KUKA KRL program: MyProgram_333().src

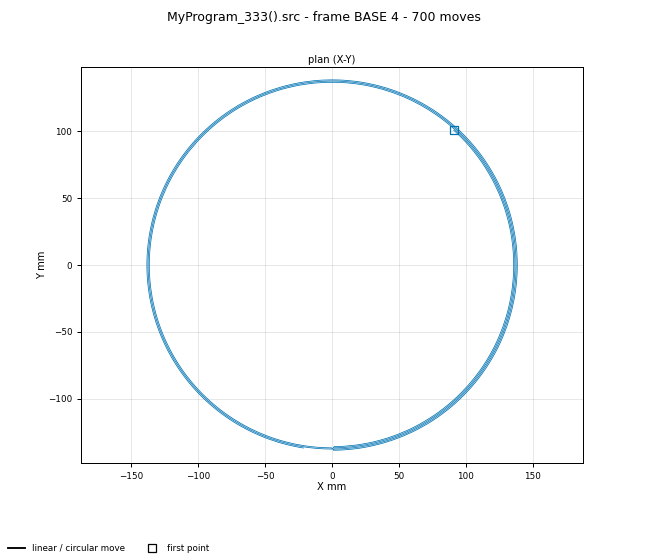
[picture p0: tool path of MyProgram_333().src in frame BASE 4, 700 of 700 moves have a stored position in this frame; points joined in program order, loops and branches not executed]
&ACCESS RVP
&REL 1
&PARAM TEMPLATE = C:\KRC\Roboter\Template\vorgabe
&PARAM EDITMASK = *
DEF MyProgram_333()
; ---- Setting reference (Base) ----
$BASE = BASE_DATA[4]

; --------------------------
; ---- Setting tool (TCP) ----
$TOOL = TOOL_DATA[3]
; --------------------------

$VEL.CP = VEL_APROX_PRINT
Startdeposition()
$VEL.CP = VEL_PRINT
LIN {X 90.8703,Y 100.8423,Z 189,A 47.7987,B 1.7183,C 0.0098,E1 1.8301,E2 406.2079} C_DIS
LIN {X 94.1895,Y 97.749,Z 189,A 46.0059,B 1.7183,C 0.013,E1 1.8337,E2 407.9863} C_DIS
LIN {X 97.3671,Y 94.5838,Z 189,A 44.2321,B 1.7183,C 0.0163,E1 1.8371,E2 409.7463} C_DIS
LIN {X 100.4728,Y 91.2777,Z 189,A 42.4362,B 1.7183,C 0.0197,E1 1.8405,E2 411.5282} C_DIS
LIN {X 103.5335,Y 87.791,Z 189,A 40.6188,B 1.7182,C 0.0232,E1 1.8438,E2 413.3292} C_DIS
LIN {X 106.2609,Y 84.4691,Z 189,A 38.9353,B 1.7182,C 0.0265,E1 1.8467,E2 414.9974} C_DIS
LIN {X 108.9996,Y 80.9045,Z 189,A 37.1372,B 1.7181,C 0.0303,E1 1.8498,E2 416.7841} C_DIS
LIN {X 111.6341,Y 77.2293,Z 189,A 34.7595,B 1.7179,C 0.0378,E1 1.8537,E2 419.2181} C_DIS
LIN {X 114.6999,Y 72.5973,Z 189,A 33.3263,B 1.7179,C 0.0378,E1 1.8557,E2 420.5428} C_DIS
LIN {X 117.6265,Y 67.7532,Z 189,A 31.0653,B 1.7179,C 0.0428,E1 1.8589,E2 422.7891} C_DIS
LIN {X 119.3923,Y 64.5914,Z 189,A 29.4618,B 1.7177,C 0.0471,E1 1.861,E2 424.4021} C_DIS
LIN {X 121.4958,Y 60.5386,Z 189,A 27.7475,B 1.7176,C 0.0506,E1 1.8632,E2 426.091} C_DIS
LIN {X 124.3864,Y 54.3522,Z 189,A 25.1966,B 1.7174,C 0.0559,E1 1.8661,E2 428.6026} C_DIS
LIN {X 125.7898,Y 51.0185,Z 189,A 23.03,B 1.7171,C 0.0642,E1 1.8685,E2 430.8476} C_DIS
LIN {X 127.7963,Y 45.7611,Z 189,A 21.5201,B 1.7171,C 0.0648,E1 1.8698,E2 432.253} C_DIS
LIN {X 128.8823,Y 42.6068,Z 189,A 20.1683,B 1.717,C 0.0681,E1 1.871,E2 433.5984} C_DIS
LIN {X 130.1919,Y 38.4196,Z 189,A 18.4533,B 1.7168,C 0.0722,E1 1.8724,E2 435.2973} C_DIS
LIN {X 131.1658,Y 34.9492,Z 189,A 17.0946,B 1.7167,C 0.0753,E1 1.8734,E2 436.6367} C_DIS
LIN {X 131.9479,Y 31.8698,Z 189,A 15.8155,B 1.7165,C 0.0785,E1 1.8743,E2 437.9086} C_DIS
LIN {X 132.7323,Y 28.4276,Z 189,A 14.4424,B 1.7164,C 0.0818,E1 1.8751,E2 439.268} C_DIS
LIN {X 133.5246,Y 24.4421,Z 189,A 12.701,B 1.7161,C 0.0867,E1 1.876,E2 441.0135} C_DIS
LIN {X 134.3255,Y 19.5645,Z 189,A 10.8763,B 1.7159,C 0.0907,E1 1.8768,E2 442.8067} C_DIS
LIN {X 135.0433,Y 13.7704,Z 189,A 8.4484,B 1.7156,C 0.0974,E1 1.8775,E2 445.2313} C_DIS
LIN {X 135.4898,Y 8.2777,Z 189,A 6.4872,B 1.7153,C 0.1014,E1 1.8779,E2 447.1481} C_DIS
LIN {X 135.6826,Y 4.0405,Z 189,A 4.2707,B 1.7149,C 0.1093,E1 1.8781,E2 449.4189} C_DIS
LIN {X 135.7388,Y -1.1337,Z 189,A 2.8572,B 1.7149,C 0.1101,E1 1.8781,E2 450.7369} C_DIS
LIN {X 135.5285,Y -7.6497,Z 189,A 0.3514,B 1.7144,C 0.1162,E1 1.8779,E2 453.2133} C_DIS
LIN {X 135.2924,Y -11.0499,Z 189,A -1.8109,B 1.7138,C 0.1252,E1 1.8774,E2 455.4679} C_DIS
LIN {X 134.6403,Y -17.266,Z 189,A -3.3061,B 1.7138,C 0.1246,E1 1.8769,E2 456.8201} C_DIS
LIN {X 134.2033,Y -20.386,Z 189,A -4.7668,B 1.7135,C 0.1292,E1 1.8763,E2 458.2983} C_DIS
LIN {X 133.5519,Y -24.2894,Z 189,A -6.2722,B 1.7132,C 0.1327,E1 1.8756,E2 459.7837} C_DIS
LIN {X 132.73,Y -28.4383,Z 189,A -7.9415,B 1.7129,C 0.1368,E1 1.8747,E2 461.4394} C_DIS
LIN {X 131.9479,Y -31.8698,Z 189,A -9.2499,B 1.7126,C 0.1397,E1 1.8739,E2 462.726} C_DIS
LIN {X 131.0873,Y -35.2437,Z 189,A -10.6477,B 1.7124,C 0.1432,E1 1.8729,E2 464.1155} C_DIS
LIN {X 130.1198,Y -38.6657,Z 189,A -12.0307,B 1.7121,C 0.1465,E1 1.8718,E2 465.4844} C_DIS
LIN {X 127.4351,Y -46.763,Z 189,A -15.4685,B 1.7113,C 0.155,E1 1.8688,E2 468.9037} C_DIS
LIN {X 124.5568,Y -53.9582,Z 189,A -18.4307,B 1.7107,C 0.1615,E1 1.8657,E2 471.8281} C_DIS
LIN {X 123.0854,Y -57.2358,Z 189,A -19.8254,B 1.7104,C 0.1646,E1 1.864,E2 473.2081} C_DIS
LIN {X 121.5338,Y -60.4615,Z 189,A -21.1963,B 1.7102,C 0.1675,E1 1.8624,E2 474.5619} C_DIS
LIN {X 119.9443,Y -63.5568,Z 189,A -22.6938,B 1.7098,C 0.1714,E1 1.8604,E2 476.0643} C_DIS
LIN {X 117.629,Y -67.7489,Z 189,A -24.6616,B 1.7093,C 0.1761,E1 1.8577,E2 478.0267} C_DIS
LIN {X 115.5415,Y -71.2508,Z 189,A -26.1596,B 1.709,C 0.1789,E1 1.8556,E2 479.4967} C_DIS
LIN {X 113.1519,Y -74.9881,Z 189,A -28.3044,B 1.7083,C 0.1852,E1 1.8523,E2 481.6786} C_DIS
LIN {X 110.5875,Y -78.7204,Z 189,A -29.805,B 1.7081,C 0.1871,E1 1.8499,E2 483.1268} C_DIS
LIN {X 106.2233,Y -84.5164,Z 189,A -32.1804,B 1.7078,C 0.1897,E1 1.8461,E2 485.4136} C_DIS
LIN {X 101.8169,Y -89.7762,Z 189,A -35.2885,B 1.7069,C 0.1975,E1 1.8404,E2 488.5522} C_DIS
LIN {X 97.0122,Y -94.9477,Z 189,A -37.7383,B 1.7066,C 0.2006,E1 1.8359,E2 490.9338} C_DIS
LIN {X 93.5191,Y -98.3907,Z 189,A -40.0626,B 1.7059,C 0.2065,E1 1.8311,E2 493.2937} C_DIS
LIN {X 89.8066,Y -101.79,Z 189,A -42.5349,B 1.7051,C 0.2129,E1 1.8258,E2 495.8137} C_DIS
LIN {X 85.9282,Y -105.0845,Z 189,A -44.0029,B 1.7051,C 0.2129,E1 1.8229,E2 497.1929} C_DIS
LIN {X 82.7199,Y -107.6287,Z 189,A -46.0103,B 1.7045,C 0.2178,E1 1.8183,E2 499.2389} C_DIS
LIN {X 79.5486,Y -109.9929,Z 189,A -47.3444,B 1.7043,C 0.2189,E1 1.8154,E2 500.5294} C_DIS
LIN {X 76.7274,Y -111.9792,Z 189,A -48.6664,B 1.7041,C 0.2206,E1 1.8124,E2 501.8344} C_DIS
LIN {X 73.1409,Y -114.354,Z 189,A -50.3736,B 1.7038,C 0.2231,E1 1.8084,E2 503.5285} C_DIS
LIN {X 66.1262,Y -118.5492,Z 189,A -53.5982,B 1.7032,C 0.2273,E1 1.8007,E2 506.7253} C_DIS
LIN {X 62.9243,Y -120.2765,Z 189,A -55.0845,B 1.703,C 0.2294,E1 1.7971,E2 508.206} C_DIS
LIN {X 59.426,Y -122.0447,Z 189,A -56.6641,B 1.7027,C 0.2313,E1 1.7931,E2 509.7766} C_DIS
LIN {X 56.28,Y -123.5274,Z 189,A -59.0747,B 1.7017,C 0.2386,E1 1.7867,E2 512.3149} C_DIS
LIN {X 49.5643,Y -126.3702,Z 189,A -60.8954,B 1.7021,C 0.2357,E1 1.7824,E2 513.9687} C_DIS
LIN {X 47.2117,Y -127.2679,Z 189,A -62.1901,B 1.7017,C 0.2382,E1 1.7789,E2 515.2956} C_DIS
LIN {X 42.7243,Y -128.8432,Z 189,A -64.0034,B 1.7016,C 0.2395,E1 1.7741,E2 517.0838} C_DIS
LIN {X 39.4837,Y -129.873,Z 189,A -65.3751,B 1.7014,C 0.2407,E1 1.7705,E2 518.4479} C_DIS
LIN {X 36.0559,Y -130.867,Z 189,A -66.9587,B 1.7011,C 0.2426,E1 1.7662,E2 520.0429} C_DIS
LIN {X 32.0339,Y -131.9083,Z 189,A -68.7073,B 1.7009,C 0.2442,E1 1.7614,E2 521.792} C_DIS
LIN {X 28.2791,Y -132.7644,Z 189,A -70.1338,B 1.7009,C 0.2446,E1 1.7576,E2 523.1924} C_DIS
LIN {X 24.9851,Y -133.424,Z 189,A -71.6086,B 1.7006,C 0.246,E1 1.7535,E2 524.6758} C_DIS
LIN {X 18.2831,Y -134.5059,Z 189,A -74.459,B 1.7004,C 0.2478,E1 1.7456,E2 527.5258} C_DIS
LIN {X 9.6151,Y -135.4017,Z 189,A -77.5536,B 1.7004,C 0.2472,E1 1.7372,E2 530.5429} C_DIS
LIN {X 5.6929,Y -135.6236,Z 189,A -80.0456,B 1.6998,C 0.2516,E1 1.7299,E2 533.1494} C_DIS
LIN {X 1.4833,Y -135.7364,Z 189,A -82.2677,B 1.6995,C 0.254,E1 1.7235,E2 535.4324} C_DIS
LIN {X 1.4833,Y -135.7364,Z 189,A -82.2677,B 1.6995,C 0.254,E1 1.7235,E2 535.4325} C_DIS
Enddeposition()
LIN {X 0.9598,Y -136.6371,Z 189,A -81.4185,B 1.6921,C 0.25,E1 1.7183,E2 534.469} C_DIS
Startdeposition()
$VEL.CP = VEL_PRINT
LIN {X 6.638,Y -136.4804,Z 189,A -78.5202,B 1.6925,C 0.2468,E1 1.7266,E2 531.4984} C_DIS
LIN {X 9.6494,Y -136.3007,Z 189,A -76.4403,B 1.6932,C 0.2424,E1 1.7327,E2 529.3043} C_DIS
LIN {X 16.0925,Y -135.6906,Z 189,A -74.9101,B 1.6926,C 0.2465,E1 1.7365,E2 527.9373} C_DIS
LIN {X 23.1959,Y -134.6601,Z 189,A -71.5532,B 1.6931,C 0.2428,E1 1.746,E2 524.531} C_DIS
LIN {X 26.9,Y -133.9678,Z 189,A -70.1444,B 1.6931,C 0.2424,E1 1.7498,E2 523.1449} C_DIS
LIN {X 30.7402,Y -133.139,Z 189,A -68.4565,B 1.6934,C 0.2408,E1 1.7544,E2 521.4504} C_DIS
LIN {X 34.9207,Y -132.104,Z 189,A -66.772,B 1.6935,C 0.2397,E1 1.7589,E2 519.7815} C_DIS
LIN {X 38.144,Y -131.2095,Z 189,A -65.4425,B 1.6937,C 0.2386,E1 1.7625,E2 518.4613} C_DIS
LIN {X 42.1979,Y -129.9638,Z 189,A -63.4142,B 1.6941,C 0.2354,E1 1.768,E2 516.3972} C_DIS
LIN {X 45.2532,Y -128.9311,Z 189,A -62.2617,B 1.6942,C 0.2349,E1 1.771,E2 515.2714} C_DIS
LIN {X 49.0394,Y -127.539,Z 189,A -60.4045,B 1.6946,C 0.2319,E1 1.7759,E2 513.3902} C_DIS
LIN {X 52.3982,Y -126.1955,Z 189,A -58.8181,B 1.6949,C 0.2296,E1 1.78,E2 511.7931} C_DIS
LIN {X 56.5287,Y -124.4023,Z 189,A -57.4744,B 1.6949,C 0.2301,E1 1.7833,E2 510.5234} C_DIS
LIN {X 60.044,Y -122.7424,Z 189,A -55.8889,B 1.6952,C 0.228,E1 1.7873,E2 508.9428} C_DIS
LIN {X 63.4072,Y -121.0385,Z 189,A -54.4087,B 1.6954,C 0.2262,E1 1.7909,E2 507.4753} C_DIS
LIN {X 67.1839,Y -118.9861,Z 189,A -52.2096,B 1.6961,C 0.2211,E1 1.7965,E2 505.2204} C_DIS
LIN {X 70.9392,Y -116.7862,Z 189,A -50.6757,B 1.6962,C 0.2198,E1 1.8,E2 503.7252} C_DIS
LIN {X 75.7995,Y -113.6916,Z 189,A -48.3467,B 1.6967,C 0.2162,E1 1.8055,E2 501.4064} C_DIS
LIN {X 78.5361,Y -111.8185,Z 189,A -47.1452,B 1.6969,C 0.2149,E1 1.8082,E2 500.2298} C_DIS
LIN {X 82.5681,Y -108.8758,Z 189,A -45.2283,B 1.6972,C 0.2121,E1 1.8124,E2 498.3355} C_DIS
LIN {X 86.127,Y -106.0833,Z 189,A -43.5538,B 1.6975,C 0.2099,E1 1.816,E2 496.6898} C_DIS
LIN {X 89.7935,Y -102.9973,Z 189,A -41.3951,B 1.6981,C 0.205,E1 1.8207,E2 494.5093} C_DIS
LIN {X 93.6526,Y -99.5014,Z 189,A -39.4677,B 1.6984,C 0.2022,E1 1.8246,E2 492.6152} C_DIS
LIN {X 96.9373,Y -96.3041,Z 189,A -37.7525,B 1.6987,C 0.1995,E1 1.8279,E2 490.9265} C_DIS
LIN {X 100.3179,Y -92.7775,Z 189,A -35.4013,B 1.6995,C 0.1931,E1 1.8325,E2 488.5326} C_DIS
LIN {X 103.1234,Y -89.649,Z 189,A -34.1162,B 1.6995,C 0.1923,E1 1.8348,E2 487.3109} C_DIS
LIN {X 105.9837,Y -86.2489,Z 189,A -32.351,B 1.7,C 0.1887,E1 1.8379,E2 485.5575} C_DIS
LIN {X 110.3626,Y -80.5696,Z 189,A -29.6513,B 1.7005,C 0.1838,E1 1.8424,E2 482.897} C_DIS
LIN {X 112.6528,Y -77.3346,Z 189,A -27.7228,B 1.7011,C 0.1781,E1 1.8455,E2 480.9314} C_DIS
LIN {X 114.7002,Y -74.2646,Z 189,A -26.5325,B 1.7013,C 0.1767,E1 1.8473,E2 479.788} C_DIS
LIN {X 117.8288,Y -69.1933,Z 189,A -24.2296,B 1.7018,C 0.1719,E1 1.8506,E2 477.5094} C_DIS
LIN {X 119.9886,Y -65.3764,Z 189,A -22.3737,B 1.7022,C 0.1671,E1 1.8531,E2 475.6498} C_DIS
LIN {X 122.2789,Y -60.9836,Z 189,A -20.5833,B 1.7026,C 0.1638,E1 1.8553,E2 473.8962} C_DIS
LIN {X 123.9248,Y -57.5629,Z 189,A -19.1561,B 1.7028,C 0.1608,E1 1.857,E2 472.4897} C_DIS
LIN {X 125.2805,Y -54.5501,Z 189,A -17.3824,B 1.7034,C 0.1545,E1 1.859,E2 470.6632} C_DIS
LIN {X 127.0806,Y -50.2186,Z 189,A -15.9513,B 1.7036,C 0.1531,E1 1.8604,E2 469.3021} C_DIS
LIN {X 128.2149,Y -47.2469,Z 189,A -13.9405,B 1.7043,C 0.1448,E1 1.8625,E2 467.2002} C_DIS
LIN {X 130.4205,Y -40.7672,Z 189,A -12.0416,B 1.7043,C 0.1439,E1 1.8639,E2 465.4285} C_DIS
LIN {X 131.5275,Y -37.0325,Z 189,A -10.6101,B 1.7046,C 0.1408,E1 1.865,E2 464.0224} C_DIS
LIN {X 132.4351,Y -33.6421,Z 189,A -9.3001,B 1.7048,C 0.1379,E1 1.8659,E2 462.7326} C_DIS
LIN {X 133.1233,Y -30.809,Z 189,A -8.0811,B 1.7051,C 0.1346,E1 1.8667,E2 461.5132} C_DIS
LIN {X 133.9655,Y -26.9115,Z 189,A -6.5538,B 1.7054,C 0.131,E1 1.8676,E2 460.0038} C_DIS
LIN {X 134.7035,Y -22.9359,Z 189,A -5.0069,B 1.7057,C 0.1273,E1 1.8683,E2 458.4751} C_DIS
LIN {X 135.245,Y -19.4862,Z 189,A -3.622,B 1.7059,C 0.1238,E1 1.8689,E2 457.0996} C_DIS
LIN {X 136.1958,Y -11.0373,Z 189,A -0.4243,B 1.7064,C 0.1165,E1 1.8698,E2 453.9476} C_DIS
LIN {X 136.4812,Y -6.6222,Z 189,A 1.7597,B 1.7069,C 0.109,E1 1.8702,E2 451.7198} C_DIS
LIN {X 136.6204,Y -2.4108,Z 189,A 2.9612,B 1.707,C 0.108,E1 1.8702,E2 450.5905} C_DIS
LIN {X 136.5503,Y 5.0048,Z 189,A 5.6575,B 1.7074,C 0.1021,E1 1.8702,E2 447.9456} C_DIS
LIN {X 136.1391,Y 11.709,Z 189,A 8.345,B 1.7078,C 0.0952,E1 1.8696,E2 445.2732} C_DIS
LIN {X 135.3864,Y 18.4923,Z 189,A 11.1821,B 1.7082,C 0.0874,E1 1.8687,E2 442.438} C_DIS
LIN {X 134.7131,Y 22.8782,Z 189,A 12.9307,B 1.7084,C 0.083,E1 1.8679,E2 440.7027} C_DIS
LIN {X 133.952,Y 26.9775,Z 189,A 14.4505,B 1.7086,C 0.0797,E1 1.8671,E2 439.2111} C_DIS
LIN {X 133.2099,Y 30.4298,Z 189,A 15.7384,B 1.7086,C 0.0769,E1 1.8664,E2 437.9468} C_DIS
LIN {X 132.5198,Y 33.3082,Z 189,A 16.9974,B 1.7088,C 0.0734,E1 1.8655,E2 436.685} C_DIS
LIN {X 131.5905,Y 36.8072,Z 189,A 18.3385,B 1.709,C 0.0705,E1 1.8646,E2 435.3655} C_DIS
LIN {X 130.5483,Y 40.3498,Z 189,A 19.8688,B 1.7091,C 0.0664,E1 1.8633,E2 433.8369} C_DIS
LIN {X 129.2766,Y 44.2566,Z 189,A 21.4331,B 1.7093,C 0.0629,E1 1.8619,E2 432.2917} C_DIS
LIN {X 126.2599,Y 52.244,Z 189,A 24.5596,B 1.7095,C 0.0565,E1 1.8589,E2 429.2208} C_DIS
LIN {X 123.4311,Y 58.6143,Z 189,A 27.4253,B 1.7097,C 0.0493,E1 1.8556,E2 426.3613} C_DIS
LIN {X 122.0152,Y 61.509,Z 189,A 28.7348,B 1.7097,C 0.0461,E1 1.854,E2 425.0566} C_DIS
LIN {X 120.1592,Y 65.0637,Z 189,A 30.359,B 1.7099,C 0.0422,E1 1.8518,E2 423.4391} C_DIS
LIN {X 118.5749,Y 67.9072,Z 189,A 31.8533,B 1.7099,C 0.038,E1 1.8497,E2 421.9283} C_DIS
LIN {X 116.6673,Y 71.1352,Z 189,A 33.075,B 1.71,C 0.0364,E1 1.848,E2 420.7496} C_DIS
LIN {X 112.8563,Y 77.0383,Z 189,A 35.8359,B 1.7101,C 0.0304,E1 1.8438,E2 418.0108} C_DIS
LIN {X 110.2059,Y 80.7838,Z 189,A 37.625,B 1.7102,C 0.0268,E1 1.8409,E2 416.2379} C_DIS
LIN {X 107.4154,Y 84.4586,Z 189,A 39.3989,B 1.7102,C 0.0233,E1 1.8379,E2 414.4833} C_DIS
LIN {X 104.6512,Y 87.8604,Z 189,A 41.1209,B 1.7103,C 0.0199,E1 1.8349,E2 412.7752} C_DIS
LIN {X 101.671,Y 91.2927,Z 189,A 42.921,B 1.7103,C 0.0163,E1 1.8316,E2 410.9877} C_DIS
LIN {X 98.5782,Y 94.6243,Z 189,A 44.7404,B 1.7103,C 0.0127,E1 1.8281,E2 409.1787} C_DIS
LIN {X 95.382,Y 97.8456,Z 189,A 46.5468,B 1.7103,C 0.0093,E1 1.8245,E2 407.3838} C_DIS
LIN {X 92.0466,Y 100.9893,Z 189,A 48.3479,B 1.7104,C 0.0061,E1 1.8209,E2 405.5971} C_DIS
LIN {X 88.6095,Y 104.0178,Z 189,A 50.136,B 1.7104,C 0.0031,E1 1.8171,E2 403.825} C_DIS
LIN {X 85.2404,Y 106.7962,Z 189,A 51.8877,B 1.7104,C 0.0001,E1 1.8133,E2 402.0828} C_DIS
LIN {X 81.552,Y 109.6385,Z 189,A 53.7124,B 1.7104,C -0.0028,E1 1.8093,E2 400.2734} C_DIS
LIN {X 77.8266,Y 112.314,Z 189,A 55.5276,B 1.7104,C -0.0056,E1 1.8052,E2 398.4712} C_DIS
LIN {X 75.274,Y 114.0403,Z 189,A 56.9875,B 1.7104,C -0.0087,E1 1.8017,E2 396.9912} C_DIS
LIN {X 72.4248,Y 115.8708,Z 189,A 58.1526,B 1.7104,C -0.0097,E1 1.799,E2 395.8567} C_DIS
LIN {X 65.461,Y 119.9425,Z 189,A 61.3619,B 1.7104,C -0.0141,E1 1.7913,E2 392.6685} C_DIS
LIN {X 62.0137,Y 121.7583,Z 189,A 62.8249,B 1.7104,C -0.0156,E1 1.7877,E2 391.2258} C_DIS
LIN {X 59.2489,Y 123.1279,Z 189,A 64.1239,B 1.7104,C -0.0175,E1 1.7844,E2 389.9264} C_DIS
LIN {X 56.0936,Y 124.5969,Z 189,A 65.9051,B 1.7103,C -0.0211,E1 1.7798,E2 388.1071} C_DIS
LIN {X 52.3794,Y 126.2033,Z 189,A 67.0714,B 1.7103,C -0.0206,E1 1.7769,E2 387.004} C_DIS
LIN {X 45.3547,Y 128.8959,Z 189,A 70.2291,B 1.7103,C -0.0244,E1 1.7686,E2 383.8468} C_DIS
LIN {X 41.7002,Y 130.1227,Z 189,A 71.7313,B 1.7103,C -0.0256,E1 1.7647,E2 382.3584} C_DIS
LIN {X 38.8235,Y 131.0105,Z 189,A 73.0287,B 1.7103,C -0.0271,E1 1.7612,E2 381.0572} C_DIS
LIN {X 35.1939,Y 132.0311,Z 189,A 74.479,B 1.7102,C -0.028,E1 1.7573,E2 379.6226} C_DIS
LIN {X 31.8893,Y 132.8681,Z 189,A 75.8705,B 1.7102,C -0.0292,E1 1.7535,E2 378.2359} C_DIS
LIN {X 28.3006,Y 133.6796,Z 189,A 77.4356,B 1.7102,C -0.0305,E1 1.7492,E2 376.6687} C_DIS
LIN {X 24.5752,Y 134.4142,Z 189,A 78.9982,B 1.7102,C -0.0316,E1 1.7449,E2 375.11} C_DIS
LIN {X 20.9792,Y 135.0213,Z 189,A 80.6075,B 1.7101,C -0.033,E1 1.7405,E2 373.4918} C_DIS
LIN {X 16.3542,Y 135.6594,Z 189,A 82.3767,B 1.7101,C -0.0334,E1 1.7356,E2 371.7453} C_DIS
LIN {X 10.763,Y 136.2189,Z 189,A 84.6514,B 1.7101,C -0.0342,E1 1.7293,E2 369.481} C_DIS
LIN {X 3.0608,Y 136.6093,Z 189,A 87.8409,B 1.7101,C -0.0353,E1 1.7204,E2 366.2981} C_DIS
LIN {X -4.6502,Y 136.5641,Z 189,A 92.1462,B 1.71,C -0.0399,E1 1.7079,E2 361.868} C_DIS
LIN {X -11.9001,Y 136.1229,Z 189,A 94.1225,B 1.71,C -0.0362,E1 1.7028,E2 360.019} C_DIS
LIN {X -16.1251,Y 135.6867,Z 189,A 95.9512,B 1.71,C -0.0362,E1 1.6977,E2 358.1857} C_DIS
LIN {X -23.2029,Y 134.6589,Z 189,A 99.0913,B 1.71,C -0.0362,E1 1.6889,E2 355.0306} C_DIS
LIN {X -27.1929,Y 133.9082,Z 189,A 100.645,B 1.71,C -0.0352,E1 1.6847,E2 353.4951} C_DIS
LIN {X -30.3392,Y 133.2306,Z 189,A 102.0319,B 1.71,C -0.0348,E1 1.6809,E2 352.1045} C_DIS
LIN {X -33.6206,Y 132.4405,Z 189,A 103.4406,B 1.71,C -0.0342,E1 1.677,E2 350.6973} C_DIS
LIN {X -36.8084,Y 131.5902,Z 189,A 104.852,B 1.71,C -0.0336,E1 1.6732,E2 349.2834} C_DIS
LIN {X -40.2075,Y 130.5918,Z 189,A 106.3833,B 1.7101,C -0.0328,E1 1.6691,E2 347.7475} C_DIS
LIN {X -46.3097,Y 128.5543,Z 189,A 109.5035,B 1.7101,C -0.0321,E1 1.6607,E2 344.5793} C_DIS
LIN {X -49.7628,Y 127.2578,Z 189,A 110.7415,B 1.7101,C -0.0301,E1 1.6576,E2 343.3785} C_DIS
LIN {X -52.5932,Y 126.114,Z 189,A 112.0559,B 1.7101,C -0.0291,E1 1.6541,E2 342.0607} C_DIS
LIN {X -57.0752,Y 124.1503,Z 189,A 114.1495,B 1.7101,C -0.0273,E1 1.6488,E2 339.9635} C_DIS
LIN {X -60.0734,Y 122.7279,Z 189,A 115.5267,B 1.7102,C -0.0259,E1 1.6453,E2 338.5889} C_DIS
LIN {X -63.2218,Y 121.1358,Z 189,A 117.0534,B 1.7102,C -0.0244,E1 1.6415,E2 337.0575} C_DIS
LIN {X -68.1531,Y 118.434,Z 189,A 119.6797,B 1.7102,C -0.0222,E1 1.635,E2 334.4012} C_DIS
LIN {X -70.9604,Y 116.7735,Z 189,A 121.4549,B 1.7102,C -0.0213,E1 1.6306,E2 332.5787} C_DIS
LIN {X -74.515,Y 114.5376,Z 189,A 122.8384,B 1.7103,C -0.0182,E1 1.6275,E2 331.241} C_DIS
LIN {X -78.0771,Y 112.1396,Z 189,A 124.5433,B 1.7103,C -0.0155,E1 1.6236,E2 329.5485} C_DIS
LIN {X -80.2964,Y 110.5614,Z 189,A 126.1401,B 1.7103,C -0.0147,E1 1.6198,E2 327.8988} C_DIS
LIN {X -86.1397,Y 106.0729,Z 189,A 129.2414,B 1.7103,C -0.0099,E1 1.613,E2 324.7982} C_DIS
LIN {X -88.7733,Y 103.8786,Z 189,A 131.3601,B 1.7103,C -0.0086,E1 1.6083,E2 322.599} C_DIS
LIN {X -92.8079,Y 100.2904,Z 189,A 133.9909,B 1.7104,C -0.0052,E1 1.6028,E2 319.9256} C_DIS
LIN {X -97.5298,Y 95.7041,Z 189,A 135.8376,B 1.7104,C 0.0013,E1 1.5994,E2 318.1905} C_DIS
LIN {X -100.9149,Y 92.1271,Z 189,A 138.3985,B 1.7104,C 0.0046,E1 1.5944,E2 315.5717} C_DIS
LIN {X -106.3102,Y 85.8457,Z 189,A 141.9258,B 1.7104,C 0.0116,E1 1.588,E2 312.0403} C_DIS
LIN {X -108.7544,Y 82.728,Z 189,A 143.756,B 1.7104,C 0.0149,E1 1.5849,E2 310.1909} C_DIS
LIN {X -111.4395,Y 79.074,Z 189,A 145.7651,B 1.7104,C 0.0189,E1 1.5816,E2 308.1701} C_DIS
LIN {X -113.8609,Y 75.5458,Z 189,A 147.6839,B 1.7103,C 0.0228,E1 1.5785,E2 306.2375} C_DIS
LIN {X -116.2536,Y 71.8096,Z 189,A 149.4367,B 1.7102,C 0.0272,E1 1.576,E2 304.499} C_DIS
LIN {X -118.0562,Y 68.8057,Z 189,A 151.3036,B 1.7102,C 0.0303,E1 1.5732,E2 302.5849} C_DIS
LIN {X -119.6676,Y 65.9626,Z 189,A 152.9471,B 1.7101,C 0.0333,E1 1.571,E2 300.9089} C_DIS
LIN {X -122.0524,Y 61.4359,Z 189,A 155.0864,B 1.71,C 0.0385,E1 1.5682,E2 298.7718} C_DIS
LIN {X -123.8591,Y 57.7048,Z 189,A 156.8248,B 1.7099,C 0.0428,E1 1.5662,E2 297.0346} C_DIS
LIN {X -125.1899,Y 54.7596,Z 189,A 158.1686,B 1.7098,C 0.0463,E1 1.5646,E2 295.6932} C_DIS
LIN {X -126.4827,Y 51.7047,Z 189,A 159.8525,B 1.7097,C 0.0496,E1 1.5628,E2 293.9743} C_DIS
LIN {X -127.7948,Y 48.3686,Z 189,A 161.4874,B 1.7096,C 0.0534,E1 1.5611,E2 292.3241} C_DIS
LIN {X -128.9938,Y 45.0723,Z 189,A 163.0488,B 1.7095,C 0.0571,E1 1.5597,E2 290.7525} C_DIS
LIN {X -130.0845,Y 41.8197,Z 189,A 164.4928,B 1.7093,C 0.0609,E1 1.5584,E2 289.3088} C_DIS
LIN {X -131.0021,Y 38.8523,Z 189,A 166.0466,B 1.7093,C 0.0642,E1 1.5571,E2 287.7247} C_DIS
LIN {X -131.8937,Y 35.7092,Z 189,A 167.4507,B 1.7091,C 0.0679,E1 1.5561,E2 286.3173} C_DIS
LIN {X -132.7764,Y 32.2699,Z 189,A 169.5327,B 1.7089,C 0.0715,E1 1.5546,E2 284.1622} C_DIS
LIN {X -133.6236,Y 28.56,Z 189,A 170.8856,B 1.7087,C 0.076,E1 1.5539,E2 282.8408} C_DIS
LIN {X -134.465,Y 24.2915,Z 189,A 172.8303,B 1.7085,C 0.081,E1 1.5528,E2 280.8822} C_DIS
LIN {X -135.0064,Y 21.0758,Z 189,A 174.3373,B 1.7083,C 0.0846,E1 1.5522,E2 279.3585} C_DIS
LIN {X -135.5131,Y 17.5257,Z 189,A 175.99,B 1.7081,C 0.0887,E1 1.5515,E2 277.688} C_DIS
LIN {X -135.9756,Y 13.4807,Z 189,A 177.8709,B 1.7079,C 0.0934,E1 1.551,E2 275.7862} C_DIS
LIN {X -136.284,Y 9.8785,Z 189,A 179.4831,B 1.7076,C 0.0975,E1 1.5506,E2 274.1627} C_DIS
LIN {X -136.5156,Y 5.8948,Z 189,A -178.5868,B 1.7074,C 0.102,E1 1.5503,E2 272.201} C_DIS
LIN {X -136.6273,Y 1.9955,Z 189,A -176.8494,B 1.7071,C 0.1066,E1 1.5503,E2 270.4516} C_DIS
LIN {X -136.6254,Y -2.1155,Z 189,A -175.0317,B 1.7068,C 0.1113,E1 1.5503,E2 268.623} C_DIS
LIN {X -136.5337,Y -5.4291,Z 189,A -173.4611,B 1.7065,C 0.1151,E1 1.5504,E2 267.0301} C_DIS
LIN {X -136.3026,Y -9.6245,Z 189,A -171.5293,B 1.7062,C 0.1199,E1 1.5508,E2 265.0774} C_DIS
LIN {X -135.9815,Y -13.4185,Z 189,A -169.71,B 1.7059,C 0.1242,E1 1.5512,E2 263.2303} C_DIS
LIN {X -135.4987,Y -17.6351,Z 189,A -167.9286,B 1.7055,C 0.1291,E1 1.5518,E2 261.4496} C_DIS
LIN {X -135.0523,Y -20.7792,Z 189,A -166.4401,B 1.7053,C 0.1327,E1 1.5525,E2 259.9416} C_DIS
LIN {X -134.5164,Y -24.0042,Z 189,A -164.9986,B 1.705,C 0.1364,E1 1.5532,E2 258.4915} C_DIS
LIN {X -133.8905,Y -27.2799,Z 189,A -163.402,B 1.7047,C 0.1401,E1 1.554,E2 256.8699} C_DIS
LIN {X -133.0557,Y -31.1049,Z 189,A -161.5924,B 1.7043,C 0.1444,E1 1.5552,E2 255.0393} C_DIS
LIN {X -132.3584,Y -33.9441,Z 189,A -160.2296,B 1.704,C 0.1476,E1 1.5561,E2 253.6591} C_DIS
LIN {X -131.2105,Y -38.1405,Z 189,A -158.2885,B 1.7036,C 0.1523,E1 1.5576,E2 251.7036} C_DIS
LIN {X -130.1243,Y -41.6952,Z 189,A -156.5897,B 1.7033,C 0.1563,E1 1.559,E2 249.987} C_DIS
LIN {X -128.9301,Y -45.2561,Z 189,A -154.289,B 1.7029,C 0.1597,E1 1.5612,E2 247.5911} C_DIS
LIN {X -127.2697,Y -49.732,Z 189,A -152.6874,B 1.7024,C 0.1652,E1 1.5628,E2 246.0434} C_DIS
LIN {X -125.5599,Y -53.9038,Z 189,A -150.6966,B 1.702,C 0.1699,E1 1.5649,E2 244.0401} C_DIS
LIN {X -124.1504,Y -57.0749,Z 189,A -149.1328,B 1.7016,C 0.1734,E1 1.5668,E2 242.4624} C_DIS
LIN {X -122.6635,Y -60.2039,Z 189,A -147.5487,B 1.7013,C 0.1768,E1 1.5687,E2 240.8614} C_DIS
LIN {X -121.1718,Y -63.1533,Z 189,A -146.0039,B 1.7009,C 0.18,E1 1.5707,E2 239.2959} C_DIS
LIN {X -118.4525,Y -68.1211,Z 189,A -143.4059,B 1.7003,C 0.1853,E1 1.5743,E2 236.669} C_DIS
LIN {X -115.9691,Y -72.267,Z 189,A -141.2118,B 1.6999,C 0.1898,E1 1.5775,E2 234.4529} C_DIS
LIN {X -113.4181,Y -76.2092,Z 189,A -139.0916,B 1.6994,C 0.1939,E1 1.5808,E2 232.3129} C_DIS
LIN {X -110.8691,Y -79.872,Z 189,A -137.1182,B 1.6989,C 0.1978,E1 1.584,E2 230.3262} C_DIS
LIN {X -108.36,Y -83.2438,Z 189,A -135.2315,B 1.6985,C 0.2014,E1 1.5873,E2 228.423} C_DIS
LIN {X -105.5156,Y -86.8214,Z 189,A -133.1565,B 1.6981,C 0.205,E1 1.5909,E2 226.3271} C_DIS
LIN {X -102.6298,Y -90.2142,Z 189,A -131.3143,B 1.6976,C 0.2088,E1 1.5943,E2 224.4885} C_DIS
LIN {X -99.9444,Y -93.1797,Z 189,A -129.4498,B 1.6973,C 0.2116,E1 1.5979,E2 222.5989} C_DIS
LIN {X -96.7887,Y -96.4536,Z 189,A -127.5097,B 1.6968,C 0.2151,E1 1.6017,E2 220.6545} C_DIS
LIN {X -92.0452,Y -100.9906,Z 189,A -124.4897,B 1.6963,C 0.2194,E1 1.6079,E2 217.5984} C_DIS
LIN {X -88.7519,Y -103.8968,Z 189,A -122.5547,B 1.6959,C 0.2222,E1 1.612,E2 215.6508} C_DIS
LIN {X -85.433,Y -106.6429,Z 189,A -120.6349,B 1.6956,C 0.2248,E1 1.6162,E2 213.7155} C_DIS
LIN {X -81.8626,Y -109.4073,Z 189,A -118.6819,B 1.6952,C 0.2275,E1 1.6206,E2 211.7543} C_DIS
LIN {X -78.7937,Y -111.6373,Z 189,A -116.324,B 1.6952,C 0.2279,E1 1.6263,E2 209.2908} C_DIS
LIN {X -73.9097,Y -114.9294,Z 189,A -113.6794,B 1.6948,C 0.2306,E1 1.6326,E2 206.6217} C_DIS
LIN {X -68.5689,Y -118.1933,Z 189,A -111.731,B 1.6941,C 0.2356,E1 1.637,E2 204.7665} C_DIS
LIN {X -64.5385,Y -120.4415,Z 189,A -109.681,B 1.6939,C 0.2375,E1 1.6421,E2 202.7005} C_DIS
LIN {X -60.7252,Y -122.4064,Z 189,A -107.9429,B 1.6936,C 0.2395,E1 1.6464,E2 200.9705} C_DIS
LIN {X -54.9218,Y -125.1197,Z 189,A -105.2484,B 1.6932,C 0.242,E1 1.6533,E2 198.2744} C_DIS
LIN {X -48.7593,Y -127.6478,Z 189,A -102.27,B 1.693,C 0.2436,E1 1.6611,E2 195.27} C_DIS
LIN {X -45.2659,Y -128.9267,Z 189,A -100.7381,B 1.6928,C 0.2447,E1 1.6652,E2 193.7414} C_DIS
LIN {X -41.8734,Y -130.0674,Z 189,A -99.2014,B 1.6928,C 0.2455,E1 1.6693,E2 192.1994} C_DIS
LIN {X -38.6322,Y -131.0666,Z 189,A -97.8234,B 1.6926,C 0.2465,E1 1.673,E2 190.8271} C_DIS
LIN {X -35.3632,Y -131.986,Z 189,A -96.3824,B 1.6925,C 0.2471,E1 1.6769,E2 189.3832} C_DIS
LIN {X -32.0203,Y -132.8365,Z 189,A -94.8891,B 1.6925,C 0.2475,E1 1.6809,E2 187.883} C_DIS
LIN {X -28.7701,Y -133.5782,Z 189,A -93.4575,B 1.6924,C 0.2479,E1 1.6849,E2 186.4462} C_DIS
LIN {X -25.8846,Y -134.1675,Z 189,A -92.0451,B 1.6924,C 0.2475,E1 1.6888,E2 185.0088} C_DIS
LIN {X -20.3962,Y -135.1116,Z 189,A -89.8823,B 1.6923,C 0.2486,E1 1.6948,E2 182.869} C_DIS
LIN {X -15.5572,Y -135.7542,Z 189,A -87.6928,B 1.6923,C 0.2482,E1 1.7009,E2 180.659} C_DIS
LIN {X -10.2679,Y -136.2556,Z 189,A -85.6107,B 1.6923,C 0.2487,E1 1.7067,E2 178.5961} C_DIS
LIN {X -6.7856,Y -136.473,Z 189,A -84.2965,B 1.6922,C 0.2492,E1 1.7103,E2 177.3018} C_DIS
LIN {X -0.4259,Y -136.6414,Z 189,A -81.4851,B 1.6923,C 0.248,E1 1.7182,E2 174.4693} C_DIS
LIN {X -0.4259,Y -136.6414,Z 189,A -81.4852,B 1.6923,C 0.248,E1 1.7182,E2 174.4695} C_DIS
Enddeposition()
LIN {X 0.9622,Y -137.536,Z 189,A -81.4048,B 1.6895,C 0.2508,E1 1.7158,E2 174.487} C_DIS
Startdeposition()
$VEL.CP = VEL_PRINT
LIN {X -2.2745,Y -137.522,Z 189,A -83.0559,B 1.6893,C 0.2524,E1 1.711,E2 176.1807} C_DIS
LIN {X -5.9519,Y -137.4132,Z 189,A -84.4823,B 1.6893,C 0.2522,E1 1.7071,E2 177.5932} C_DIS
LIN {X -10.1341,Y -137.1669,Z 189,A -86.0573,B 1.6893,C 0.2516,E1 1.7027,E2 179.1455} C_DIS
LIN {X -13.4494,Y -136.8819,Z 189,A -87.4663,B 1.6893,C 0.2518,E1 1.6988,E2 180.5583} C_DIS
LIN {X -17.0408,Y -136.4828,Z 189,A -89.3316,B 1.6892,C 0.2531,E1 1.6935,E2 182.4739} C_DIS
LIN {X -20.4871,Y -136.0074,Z 189,A -90.5284,B 1.6893,C 0.2519,E1 1.6902,E2 183.6365} C_DIS
LIN {X -26.868,Y -134.8919,Z 189,A -93.0601,B 1.6895,C 0.2507,E1 1.6833,E2 186.1462} C_DIS
LIN {X -30.8595,Y -134.034,Z 189,A -94.8556,B 1.6895,C 0.2505,E1 1.6783,E2 187.9554} C_DIS
LIN {X -34.0149,Y -133.2681,Z 189,A -96.245,B 1.6896,C 0.2501,E1 1.6745,E2 189.3503} C_DIS
LIN {X -37.2944,Y -132.3879,Z 189,A -97.7206,B 1.6896,C 0.2496,E1 1.6705,E2 190.8347} C_DIS
LIN {X -41.4593,Y -131.1436,Z 189,A -99.6421,B 1.6898,C 0.249,E1 1.6653,E2 192.7721} C_DIS
LIN {X -45.1489,Y -129.9189,Z 189,A -101.1766,B 1.69,C 0.2476,E1 1.6613,E2 194.2952} C_DIS
LIN {X -48.7806,Y -128.6006,Z 189,A -102.8362,B 1.6901,C 0.2467,E1 1.6569,E2 195.9622} C_DIS
LIN {X -53.7498,Y -126.6054,Z 189,A -105.1092,B 1.6904,C 0.245,E1 1.651,E2 198.2416} C_DIS
LIN {X -57.2786,Y -125.0469,Z 189,A -106.9476,B 1.6904,C 0.2442,E1 1.6462,E2 200.1121} C_DIS
LIN {X -61.1071,Y -123.2206,Z 189,A -108.6006,B 1.6908,C 0.2422,E1 1.6421,E2 201.7497} C_DIS
LIN {X -64.666,Y -121.3931,Z 189,A -110.4044,B 1.691,C 0.2408,E1 1.6376,E2 203.5726} C_DIS
LIN {X -68.444,Y -119.3038,Z 189,A -112.261,B 1.6912,C 0.2389,E1 1.633,E2 205.4375} C_DIS
LIN {X -73.0531,Y -116.5388,Z 189,A -114.5529,B 1.6916,C 0.2362,E1 1.6275,E2 207.7369} C_DIS
LIN {X -76.6885,Y -114.1792,Z 189,A -116.6732,B 1.6918,C 0.2346,E1 1.6225,E2 209.9003} C_DIS
LIN {X -79.3491,Y -112.3458,Z 189,A -117.7564,B 1.6922,C 0.2321,E1 1.6201,E2 210.9476} C_DIS
LIN {X -82.5116,Y -110.0449,Z 189,A -119.6123,B 1.6924,C 0.2302,E1 1.6158,E2 212.8345} C_DIS
LIN {X -86.0443,Y -107.3051,Z 189,A -121.5577,B 1.6928,C 0.2275,E1 1.6115,E2 214.7912} C_DIS
LIN {X -89.536,Y -104.4091,Z 189,A -123.5507,B 1.6932,C 0.2247,E1 1.6072,E2 216.7981} C_DIS
LIN {X -93.0329,Y -101.3052,Z 189,A -125.694,B 1.6936,C 0.2218,E1 1.6027,E2 218.9679} C_DIS
LIN {X -96.703,Y -97.8085,Z 189,A -127.82,B 1.6941,C 0.218,E1 1.5984,E2 221.0956} C_DIS
LIN {X -99.7731,Y -94.675,Z 189,A -129.7789,B 1.6945,C 0.2149,E1 1.5946,E2 223.0721} C_DIS
LIN {X -102.8599,Y -91.3115,Z 189,A -131.737,B 1.6949,C 0.2113,E1 1.5909,E2 225.0375} C_DIS
LIN {X -105.6925,Y -88.0177,Z 189,A -133.724,B 1.6953,C 0.208,E1 1.5873,E2 227.0481} C_DIS
LIN {X -108.547,Y -84.4718,Z 189,A -135.7365,B 1.6958,C 0.2042,E1 1.5837,E2 229.0759} C_DIS
LIN {X -111.3516,Y -80.7384,Z 189,A -137.7789,B 1.6962,C 0.2002,E1 1.5803,E2 231.1308} C_DIS
LIN {X -113.9886,Y -76.9707,Z 189,A -139.8175,B 1.6967,C 0.1962,E1 1.5771,E2 233.1854} C_DIS
LIN {X -116.3495,Y -73.353,Z 189,A -141.7747,B 1.6972,C 0.1924,E1 1.5741,E2 235.1632} C_DIS
LIN {X -117.8984,Y -70.8378,Z 189,A -143.1025,B 1.6975,C 0.1897,E1 1.5721,E2 236.5037} C_DIS
LIN {X -121.9308,Y -63.6419,Z 189,A -146.6706,B 1.6983,C 0.1817,E1 1.5673,E2 240.0882} C_DIS
LIN {X -123.4778,Y -60.5857,Z 189,A -148.229,B 1.6987,C 0.1784,E1 1.5653,E2 241.6635} C_DIS
LIN {X -125.0341,Y -57.3062,Z 189,A -149.8516,B 1.6991,C 0.1747,E1 1.5634,E2 243.3002} C_DIS
LIN {X -126.5323,Y -53.9204,Z 189,A -151.5118,B 1.6994,C 0.171,E1 1.5615,E2 244.9754} C_DIS
LIN {X -127.7979,Y -50.8469,Z 189,A -153.2838,B 1.6998,C 0.1679,E1 1.5596,E2 246.7979} C_DIS
LIN {X -129.5367,Y -46.2359,Z 189,A -155.2429,B 1.7003,C 0.1625,E1 1.5577,E2 248.7438} C_DIS
LIN {X -130.5078,Y -43.4172,Z 189,A -156.6165,B 1.7006,C 0.1593,E1 1.5565,E2 250.1341} C_DIS
LIN {X -131.5889,Y -40.0221,Z 189,A -158.2118,B 1.7009,C 0.1555,E1 1.5552,E2 251.7433} C_DIS
LIN {X -132.544,Y -36.7362,Z 189,A -159.6937,B 1.7013,C 0.1518,E1 1.554,E2 253.232} C_DIS
LIN {X -133.3643,Y -33.6359,Z 189,A -161.23,B 1.7016,C 0.1484,E1 1.5529,E2 254.7937} C_DIS
LIN {X -134.3263,Y -29.5659,Z 189,A -163.194,B 1.702,C 0.1438,E1 1.5517,E2 256.7857} C_DIS
LIN {X -135.1548,Y -25.5087,Z 189,A -164.9236,B 1.7023,C 0.1391,E1 1.5507,E2 258.515} C_DIS
LIN {X -135.7142,Y -22.3417,Z 189,A -166.3846,B 1.7026,C 0.1355,E1 1.55,E2 259.991} C_DIS
LIN {X -136.1327,Y -19.6299,Z 189,A -167.7094,B 1.7029,C 0.1325,E1 1.5495,E2 261.3387} C_DIS
LIN {X -136.5877,Y -16.163,Z 189,A -169.3275,B 1.7032,C 0.1286,E1 1.5489,E2 262.9767} C_DIS
LIN {X -136.9828,Y -12.398,Z 189,A -171.1325,B 1.7035,C 0.1243,E1 1.5484,E2 264.8102} C_DIS
LIN {X -137.283,Y -8.4164,Z 189,A -172.8067,B 1.7038,C 0.1197,E1 1.5481,E2 266.4848} C_DIS
LIN {X -137.4484,Y -5.0497,Z 189,A -174.4031,B 1.7041,C 0.1159,E1 1.5479,E2 268.105} C_DIS
LIN {X -137.5398,Y -0.7491,Z 189,A -176.3603,B 1.7044,C 0.111,E1 1.5479,E2 270.0821} C_DIS
LIN {X -137.4966,Y 3.499,Z 189,A -178.3177,B 1.7047,C 0.1062,E1 1.5479,E2 272.0623} C_DIS
LIN {X -137.3539,Y 7.1724,Z 189,A -179.9171,B 1.705,C 0.1019,E1 1.5481,E2 273.6694} C_DIS
LIN {X -137.0783,Y 11.2728,Z 189,A 178.158,B 1.7053,C 0.0973,E1 1.5485,E2 275.6201} C_DIS
LIN {X -136.671,Y 15.4607,Z 189,A 176.111,B 1.7055,C 0.0926,E1 1.5491,E2 277.703} C_DIS
LIN {X -136.1566,Y 19.463,Z 189,A 174.4521,B 1.7058,C 0.0879,E1 1.5498,E2 279.358} C_DIS
LIN {X -135.6586,Y 22.6748,Z 189,A 172.9664,B 1.7059,C 0.0842,E1 1.5504,E2 280.8593} C_DIS
LIN {X -135.0148,Y 26.2408,Z 189,A 171.3006,B 1.7061,C 0.0802,E1 1.5513,E2 282.5437} C_DIS
LIN {X -134.0749,Y 30.6807,Z 189,A 169.3626,B 1.7064,C 0.0751,E1 1.5525,E2 284.4863} C_DIS
LIN {X -133.3455,Y 33.71,Z 189,A 167.7802,B 1.7065,C 0.0717,E1 1.5535,E2 286.1032} C_DIS
LIN {X -132.258,Y 37.7589,Z 189,A 165.7706,B 1.7067,C 0.0672,E1 1.5551,E2 288.1442} C_DIS
LIN {X -130.8956,Y 42.2357,Z 189,A 163.8287,B 1.7069,C 0.062,E1 1.5567,E2 290.0838} C_DIS
LIN {X -129.9052,Y 45.1884,Z 189,A 162.4298,B 1.707,C 0.0587,E1 1.5579,E2 291.4943} C_DIS
LIN {X -128.7128,Y 48.4811,Z 189,A 160.8388,B 1.7071,C 0.055,E1 1.5595,E2 293.1006} C_DIS
LIN {X -127.3218,Y 52.0279,Z 189,A 159.1443,B 1.7073,C 0.051,E1 1.5613,E2 294.8071} C_DIS
LIN {X -126.0124,Y 55.1228,Z 189,A 157.636,B 1.7073,C 0.0476,E1 1.5629,E2 296.3278} C_DIS
LIN {X -124.6195,Y 58.2029,Z 189,A 156.0165,B 1.7075,C 0.0442,E1 1.5649,E2 297.9721} C_DIS
LIN {X -123.2527,Y 61.042,Z 189,A 154.6535,B 1.7075,C 0.041,E1 1.5666,E2 299.3402} C_DIS
LIN {X -121.3396,Y 64.7666,Z 189,A 152.6234,B 1.7076,C 0.037,E1 1.5692,E2 301.4038} C_DIS
LIN {X -119.1222,Y 68.759,Z 189,A 150.3547,B 1.7077,C 0.0329,E1 1.5724,E2 303.7153} C_DIS
LIN {X -117.2752,Y 71.8638,Z 189,A 149.2793,B 1.7077,C 0.0289,E1 1.5739,E2 304.738} C_DIS
LIN {X -115.58,Y 74.5607,Z 189,A 147.5783,B 1.7078,C 0.0263,E1 1.5765,E2 306.4831} C_DIS
LIN {X -113.1542,Y 78.1933,Z 189,A 145.6391,B 1.7078,C 0.0223,E1 1.5796,E2 308.4355} C_DIS
LIN {X -110.5767,Y 81.7975,Z 189,A 143.523,B 1.7079,C 0.0186,E1 1.5831,E2 310.5826} C_DIS
LIN {X -107.8408,Y 85.3719,Z 189,A 141.2055,B 1.7079,C 0.0152,E1 1.5872,E2 312.9513} C_DIS
LIN {X -104.9916,Y 88.8522,Z 189,A 139.6379,B 1.7079,C 0.011,E1 1.59,E2 314.4813} C_DIS
LIN {X -102.5217,Y 91.6906,Z 189,A 137.318,B 1.7079,C 0.0089,E1 1.5945,E2 316.889} C_DIS
LIN {X -98.6756,Y 95.8177,Z 189,A 135.5172,B 1.708,C 0.0037,E1 1.5978,E2 318.6235} C_DIS
LIN {X -95.4522,Y 99.0294,Z 189,A 133.4889,B 1.708,C 0.0004,E1 1.6019,E2 320.6662} C_DIS
LIN {X -91.4497,Y 102.737,Z 189,A 130.5505,B 1.708,C -0.0025,E1 1.6082,E2 323.6812} C_DIS
LIN {X -87.6707,Y 105.9798,Z 189,A 129.2092,B 1.708,C -0.0071,E1 1.6109,E2 324.9351} C_DIS
LIN {X -82.1983,Y 110.2783,Z 189,A 125.4066,B 1.708,C -0.01,E1 1.6195,E2 328.8418} C_DIS
LIN {X -78.4648,Y 112.9653,Z 189,A 123.8794,B 1.708,C -0.0135,E1 1.6229,E2 330.3225} C_DIS
LIN {X -74.6195,Y 115.5418,Z 189,A 121.7976,B 1.708,C -0.0158,E1 1.6278,E2 332.4209} C_DIS
LIN {X -70.6782,Y 117.9938,Z 189,A 119.8947,B 1.708,C -0.0183,E1 1.6324,E2 334.3191} C_DIS
LIN {X -67.1557,Y 120.0335,Z 189,A 118.0552,B 1.708,C -0.02,E1 1.6369,E2 336.1743} C_DIS
LIN {X -63.6703,Y 121.9159,Z 189,A 116.4535,B 1.7079,C -0.022,E1 1.6409,E2 337.7693} C_DIS
LIN {X -60.7059,Y 123.4185,Z 189,A 115.0479,B 1.7079,C -0.0234,E1 1.6444,E2 339.1765} C_DIS
LIN {X -57.7771,Y 124.8163,Z 189,A 113.5762,B 1.7079,C -0.0244,E1 1.6482,E2 340.6613} C_DIS
LIN {X -51.8324,Y 127.4006,Z 189,A 110.9362,B 1.7079,C -0.027,E1 1.6549,E2 343.2927} C_DIS
LIN {X -48.4248,Y 128.7339,Z 189,A 108.2939,B 1.7079,C -0.0252,E1 1.6622,E2 346.0628} C_DIS
LIN {X -41.7334,Y 131.0561,Z 189,A 106.2953,B 1.7078,C -0.0297,E1 1.6672,E2 347.9506} C_DIS
LIN {X -37.9359,Y 132.2073,Z 189,A 104.645,B 1.7078,C -0.0306,E1 1.6717,E2 349.5997} C_DIS
LIN {X -35.1394,Y 132.9762,Z 189,A 103.3777,B 1.7078,C -0.0311,E1 1.6751,E2 350.8732} C_DIS
LIN {X -31.4082,Y 133.9087,Z 189,A 101.7999,B 1.7078,C -0.0318,E1 1.6794,E2 352.4474} C_DIS
LIN {X -28.925,Y 134.4646,Z 189,A 100.705,B 1.7078,C -0.0321,E1 1.6824,E2 353.5457} C_DIS
LIN {X -25.3958,Y 135.1763,Z 189,A 99.0838,B 1.7078,C -0.0321,E1 1.6869,E2 355.1803} C_DIS
LIN {X -20.012,Y 136.0781,Z 189,A 96.473,B 1.7078,C -0.0315,E1 1.6943,E2 357.8287} C_DIS
LIN {X -16.0915,Y 136.5962,Z 189,A 95.286,B 1.7078,C -0.0331,E1 1.6974,E2 358.9619} C_DIS
LIN {X -12.9621,Y 136.9286,Z 189,A 93.9712,B 1.7078,C -0.0331,E1 1.7011,E2 360.2766} C_DIS
LIN {X -9.2632,Y 137.2305,Z 189,A 91.8358,B 1.7078,C -0.031,E1 1.7073,E2 362.4793} C_DIS
LIN {X -4.5445,Y 137.4676,Z 189,A 90.4858,B 1.7078,C -0.033,E1 1.7108,E2 363.7573} C_DIS
LIN {X -1.6534,Y 137.5323,Z 189,A 88.7696,B 1.7078,C -0.0308,E1 1.7158,E2 365.532} C_DIS
LIN {X 2.5107,Y 137.5181,Z 189,A 87.5765,B 1.7078,C -0.0324,E1 1.719,E2 366.6618} C_DIS
LIN {X 5.6794,Y 137.4238,Z 189,A 86.1497,B 1.7078,C -0.0315,E1 1.723,E2 368.1005} C_DIS
LIN {X 9.8368,Y 137.1886,Z 189,A 84.3436,B 1.7078,C -0.0305,E1 1.7281,E2 369.9142} C_DIS
LIN {X 15.1294,Y 136.7066,Z 189,A 82.3218,B 1.7078,C -0.0301,E1 1.7337,E2 371.913} C_DIS
LIN {X 18.4294,Y 136.3015,Z 189,A 80.357,B 1.7078,C -0.0268,E1 1.7393,E2 373.9444} C_DIS
LIN {X 23.4352,Y 135.5317,Z 189,A 78.8985,B 1.7078,C -0.0281,E1 1.7431,E2 375.327} C_DIS
LIN {X 27.1818,Y 134.828,Z 189,A 77.2776,B 1.7078,C -0.0268,E1 1.7476,E2 376.9512} C_DIS
LIN {X 30.844,Y 134.0376,Z 189,A 75.8369,B 1.7078,C -0.026,E1 1.7515,E2 378.3775} C_DIS
LIN {X 34.0155,Y 133.268,Z 189,A 74.4555,B 1.7078,C -0.0247,E1 1.7553,E2 379.7611} C_DIS
LIN {X 37.3088,Y 132.3839,Z 189,A 73.1677,B 1.7078,C -0.0239,E1 1.7587,E2 381.033} C_DIS
LIN {X 40.2399,Y 131.5222,Z 189,A 71.8638,B 1.7078,C -0.0224,E1 1.7622,E2 382.3403} C_DIS
LIN {X 43.5374,Y 130.4678,Z 189,A 70.4453,B 1.7078,C -0.021,E1 1.766,E2 383.7557} C_DIS
LIN {X 47.3834,Y 129.1227,Z 189,A 68.5814,B 1.7079,C -0.0182,E1 1.771,E2 385.6388} C_DIS
LIN {X 50.8904,Y 127.7804,Z 189,A 67.255,B 1.7079,C -0.0174,E1 1.7744,E2 386.9372} C_DIS
LIN {X 54.7092,Y 126.1913,Z 189,A 65.6333,B 1.7079,C -0.0157,E1 1.7785,E2 388.5466} C_DIS
LIN {X 58.0982,Y 124.6679,Z 189,A 64.1555,B 1.7079,C -0.0139,E1 1.7822,E2 390.0159} C_DIS
LIN {X 61.2121,Y 123.1688,Z 189,A 62.8074,B 1.7079,C -0.0123,E1 1.7856,E2 391.3531} C_DIS
LIN {X 64.7847,Y 121.3299,Z 189,A 61.0777,B 1.7079,C -0.0096,E1 1.7899,E2 393.0893} C_DIS
LIN {X 69.6319,Y 118.614,Z 189,A 59.1222,B 1.708,C -0.0078,E1 1.7946,E2 395.0022} C_DIS
LIN {X 72.381,Y 116.9571,Z 189,A 57.5886,B 1.708,C -0.0046,E1 1.7983,E2 396.559} C_DIS
LIN {X 76.2143,Y 114.4958,Z 189,A 55.8089,B 1.708,C -0.002,E1 1.8024,E2 398.3246} C_DIS
LIN {X 79.9298,Y 111.9335,Z 189,A 54.0517,B 1.708,C 0.0006,E1 1.8064,E2 400.0672} C_DIS
LIN {X 83.4743,Y 109.3157,Z 189,A 52.2919,B 1.708,C 0.0036,E1 1.8103,E2 401.818} C_DIS
LIN {X 86.9692,Y 106.5562,Z 189,A 50.5374,B 1.708,C 0.0065,E1 1.8141,E2 403.5606} C_DIS
LIN {X 90.4114,Y 103.6516,Z 189,A 48.7663,B 1.708,C 0.0096,E1 1.8179,E2 405.3192} C_DIS
LIN {X 93.7294,Y 100.6612,Z 189,A 47.0147,B 1.708,C 0.0127,E1 1.8215,E2 407.0578} C_DIS
LIN {X 96.9607,Y 97.5525,Z 189,A 45.2523,B 1.708,C 0.016,E1 1.825,E2 408.8077} C_DIS
LIN {X 100.2157,Y 94.2058,Z 189,A 43.4237,B 1.708,C 0.0195,E1 1.8285,E2 410.6226} C_DIS
LIN {X 103.0205,Y 91.1298,Z 189,A 41.794,B 1.7079,C 0.0226,E1 1.8315,E2 412.2399} C_DIS
LIN {X 106.0145,Y 87.6288,Z 189,A 39.9908,B 1.7079,C 0.0262,E1 1.8347,E2 414.0294} C_DIS
LIN {X 108.7673,Y 84.1875,Z 189,A 38.3106,B 1.7078,C 0.0295,E1 1.8376,E2 415.691} C_DIS
LIN {X 111.381,Y 80.6978,Z 189,A 36.5827,B 1.7078,C 0.0332,E1 1.8405,E2 417.4086} C_DIS
LIN {X 114.0037,Y 76.9484,Z 189,A 34.7082,B 1.7076,C 0.0375,E1 1.8434,E2 419.2797} C_DIS
LIN {X 116.1265,Y 73.7063,Z 189,A 33.2566,B 1.7076,C 0.0404,E1 1.8456,E2 420.7118} C_DIS
LIN {X 118.562,Y 69.7204,Z 189,A 31.4071,B 1.7074,C 0.0446,E1 1.8482,E2 422.55} C_DIS
LIN {X 120.9529,Y 65.4863,Z 189,A 29.5579,B 1.7074,C 0.0485,E1 1.8507,E2 424.3782} C_DIS
LIN {X 122.9438,Y 61.6669,Z 189,A 28.0089,B 1.7072,C 0.0515,E1 1.8526,E2 425.8976} C_DIS
LIN {X 124.5191,Y 58.42,Z 189,A 26.3457,B 1.7071,C 0.0564,E1 1.8546,E2 427.581} C_DIS
LIN {X 125.8806,Y 55.426,Z 189,A 25.3387,B 1.7071,C 0.0576,E1 1.8557,E2 428.5436} C_DIS
LIN {X 127.0546,Y 52.6743,Z 189,A 24.1628,B 1.707,C 0.0604,E1 1.857,E2 429.7111} C_DIS
LIN {X 128.4043,Y 49.2951,Z 189,A 22.528,B 1.7068,C 0.0652,E1 1.8587,E2 431.3613} C_DIS
LIN {X 130.0513,Y 44.7671,Z 189,A 20.9338,B 1.7067,C 0.0678,E1 1.8601,E2 432.9048} C_DIS
LIN {X 131.1436,Y 41.4593,Z 189,A 19.5661,B 1.7065,C 0.0711,E1 1.8613,E2 434.2627} C_DIS
LIN {X 132.0652,Y 38.4212,Z 189,A 18.3584,B 1.7065,C 0.0739,E1 1.8622,E2 435.4567} C_DIS
LIN {X 132.9431,Y 35.2639,Z 189,A 17.0559,B 1.7063,C 0.0772,E1 1.8632,E2 436.7518} C_DIS
LIN {X 133.9735,Y 31.1248,Z 189,A 15.3264,B 1.7061,C 0.0817,E1 1.8643,E2 438.4763} C_DIS
LIN {X 134.8234,Y 27.2049,Z 189,A 13.9047,B 1.7059,C 0.0846,E1 1.8651,E2 439.8673} C_DIS
LIN {X 135.5213,Y 23.4932,Z 189,A 12.1928,B 1.7057,C 0.0899,E1 1.866,E2 441.5976} C_DIS
LIN {X 136.1547,Y 19.4763,Z 189,A 10.6121,B 1.7054,C 0.0939,E1 1.8666,E2 443.1648} C_DIS
LIN {X 136.5788,Y 16.2377,Z 189,A 9.3031,B 1.7052,C 0.0973,E1 1.867,E2 444.4679} C_DIS
LIN {X 136.9625,Y 12.609,Z 189,A 8.1754,B 1.7052,C 0.0988,E1 1.8673,E2 445.5467} C_DIS
LIN {X 137.4202,Y 5.7733,Z 189,A 5.7263,B 1.7049,C 0.104,E1 1.8677,E2 447.9457} C_DIS
LIN {X 137.5355,Y -1.3823,Z 189,A 2.864,B 1.7044,C 0.1116,E1 1.8678,E2 450.7946} C_DIS
LIN {X 137.3839,Y -6.5751,Z 189,A 0.9669,B 1.7041,C 0.1158,E1 1.8677,E2 452.6585} C_DIS
LIN {X 137.1936,Y -9.7684,Z 189,A -0.437,B 1.7038,C 0.12,E1 1.8674,E2 454.0725} C_DIS
LIN {X 136.8745,Y -13.5261,Z 189,A -1.8338,B 1.7036,C 0.1232,E1 1.867,E2 455.4477} C_DIS
LIN {X 136.4759,Y -17.0982,Z 189,A -3.6693,B 1.7031,C 0.1297,E1 1.8664,E2 457.328} C_DIS
LIN {X 135.9043,Y -21.153,Z 189,A -4.6914,B 1.7031,C 0.1297,E1 1.866,E2 458.2626} C_DIS
LIN {X 135.4026,Y -24.1564,Z 189,A -5.9927,B 1.7028,C 0.1334,E1 1.8654,E2 459.569} C_DIS
LIN {X 134.7398,Y -27.6156,Z 189,A -7.3885,B 1.7025,C 0.137,E1 1.8647,E2 460.9565} C_DIS
LIN {X 133.9919,Y -31.044,Z 189,A -8.7009,B 1.7023,C 0.1399,E1 1.8639,E2 462.2504} C_DIS
LIN {X 133.1569,Y -34.4532,Z 189,A -10.1781,B 1.7019,C 0.1441,E1 1.8628,E2 463.7306} C_DIS
LIN {X 132.0539,Y -38.46,Z 189,A -11.7,B 1.7017,C 0.1473,E1 1.8617,E2 465.2262} C_DIS
LIN {X 130.8479,Y -42.3847,Z 189,A -13.522,B 1.7012,C 0.1527,E1 1.8602,E2 467.0641} C_DIS
LIN {X 129.7679,Y -45.5845,Z 189,A -14.528,B 1.7011,C 0.1537,E1 1.8593,E2 468.0185} C_DIS
LIN {X 128.6761,Y -48.5789,Z 189,A -15.8203,B 1.7008,C 0.157,E1 1.858,E2 469.307} C_DIS
LIN {X 127.1828,Y -52.3673,Z 189,A -17.5769,B 1.7003,C 0.1618,E1 1.8562,E2 471.0729} C_DIS
LIN {X 125.4339,Y -56.4246,Z 189,A -19.0897,B 1.7001,C 0.1644,E1 1.8545,E2 472.5437} C_DIS
LIN {X 123.7854,Y -59.9587,Z 189,A -20.5637,B 1.6998,C 0.1676,E1 1.8528,E2 473.999} C_DIS
LIN {X 122.2156,Y -63.0973,Z 189,A -22.0279,B 1.6994,C 0.1713,E1 1.8509,E2 475.4646} C_DIS
LIN {X 120.3572,Y -66.5735,Z 189,A -23.517,B 1.6991,C 0.1744,E1 1.8489,E2 476.9346} C_DIS
LIN {X 118.2621,Y -70.2282,Z 189,A -25.5942,B 1.6984,C 0.1809,E1 1.8459,E2 479.056} C_DIS
LIN {X 115.8173,Y -74.1905,Z 189,A -27.6858,B 1.6978,C 0.1866,E1 1.8427,E2 481.1692} C_DIS
LIN {X 112.2827,Y -79.4387,Z 189,A -29.7523,B 1.6975,C 0.1891,E1 1.8395,E2 483.1621} C_DIS
LIN {X 109.9265,Y -82.6685,Z 189,A -31.0461,B 1.6974,C 0.1906,E1 1.8375,E2 484.4074} C_DIS
LIN {X 107.7456,Y -85.4915,Z 189,A -32.4078,B 1.6971,C 0.1932,E1 1.8351,E2 485.7536} C_DIS
LIN {X 104.9712,Y -88.8762,Z 189,A -34.1198,B 1.6967,C 0.1966,E1 1.8321,E2 487.4521} C_DIS
LIN {X 102.0923,Y -92.1692,Z 189,A -35.8794,B 1.6963,C 0.2002,E1 1.8288,E2 489.2047} C_DIS
LIN {X 99.271,Y -95.2008,Z 189,A -37.3781,B 1.696,C 0.2024,E1 1.826,E2 490.6741} C_DIS
LIN {X 96.3896,Y -98.1168,Z 189,A -39.0503,B 1.6956,C 0.2058,E1 1.8227,E2 492.3429} C_DIS
LIN {X 93.1708,Y -101.1785,Z 189,A -40.7934,B 1.6952,C 0.2089,E1 1.8192,E2 494.0728} C_DIS
LIN {X 89.7806,Y -104.1984,Z 189,A -42.5406,B 1.6948,C 0.2118,E1 1.8155,E2 495.8018} C_DIS
LIN {X 86.6472,Y -106.8188,Z 189,A -44.2223,B 1.6944,C 0.2149,E1 1.8119,E2 497.4821} C_DIS
LIN {X 83.0767,Y -109.6185,Z 189,A -45.9992,B 1.6941,C 0.2178,E1 1.808,E2 499.2451} C_DIS
LIN {X 79.4936,Y -112.244,Z 189,A -47.7475,B 1.6937,C 0.2205,E1 1.8041,E2 500.9809} C_DIS
LIN {X 75.1028,Y -115.228,Z 189,A -49.8517,B 1.6933,C 0.2237,E1 1.7992,E2 503.0721} C_DIS
LIN {X 71.3465,Y -117.5908,Z 189,A -51.6027,B 1.693,C 0.2262,E1 1.795,E2 504.811} C_DIS
LIN {X 65.4643,Y -120.9647,Z 189,A -54.326,B 1.6925,C 0.23,E1 1.7884,E2 507.5226} C_DIS
LIN {X 62.1219,Y -122.7121,Z 189,A -55.7229,B 1.6923,C 0.2313,E1 1.785,E2 508.8967} C_DIS
LIN {X 58.8861,Y -124.2978,Z 189,A -57.3431,B 1.6919,C 0.2341,E1 1.7809,E2 510.5343} C_DIS
LIN {X 55.0823,Y -126.03,Z 189,A -59.5974,B 1.6912,C 0.2393,E1 1.7749,E2 512.8599} C_DIS
LIN {X 49.5056,Y -128.3224,Z 189,A -61.2493,B 1.6914,C 0.2378,E1 1.7709,E2 514.3959} C_DIS
LIN {X 45.915,Y -129.6525,Z 189,A -62.7927,B 1.6912,C 0.2394,E1 1.7668,E2 515.9333} C_DIS
LIN {X 43.1182,Y -130.6074,Z 189,A -63.9871,B 1.691,C 0.2406,E1 1.7637,E2 517.1234} C_DIS
LIN {X 39.9527,Y -131.6102,Z 189,A -65.3293,B 1.6908,C 0.2418,E1 1.7601,E2 518.4609} C_DIS
LIN {X 36.0714,Y -132.7277,Z 189,A -67.0609,B 1.6905,C 0.2438,E1 1.7554,E2 520.2004} C_DIS
LIN {X 32.3004,Y -133.6939,Z 189,A -68.5886,B 1.6904,C 0.2448,E1 1.7513,E2 521.7161} C_DIS
LIN {X 28.3478,Y -134.5892,Z 189,A -70.4984,B 1.69,C 0.2473,E1 1.746,E2 523.6575} C_DIS
LIN {X 24.9409,Y -135.2622,Z 189,A -71.5532,B 1.6901,C 0.2465,E1 1.7432,E2 524.6591} C_DIS
LIN {X 21.7265,Y -135.8155,Z 189,A -73.493,B 1.6896,C 0.2503,E1 1.7376,E2 526.6798} C_DIS
LIN {X 16.9352,Y -136.4956,Z 189,A -75.2189,B 1.6896,C 0.2502,E1 1.7329,E2 528.367} C_DIS
LIN {X 13.5864,Y -136.8687,Z 189,A -76.5909,B 1.6896,C 0.2508,E1 1.7291,E2 529.7354} C_DIS
LIN {X 10.257,Y -137.1579,Z 189,A -77.656,B 1.6896,C 0.25,E1 1.7262,E2 530.7561} C_DIS
LIN {X 6.8165,Y -137.3718,Z 189,A -79.1161,B 1.6896,C 0.2507,E1 1.7221,E2 532.2203} C_DIS
LIN {X 1.5165,Y -137.5345,Z 189,A -81.3749,B 1.6894,C 0.2516,E1 1.7158,E2 534.4872} C_DIS
LIN {X 1.5165,Y -137.5345,Z 189,A -81.3749,B 1.6894,C 0.2516,E1 1.7158,E2 534.4872} C_DIS
Enddeposition()
LIN {X 0.9672,Y -138.4367,Z 189,A -81.2272,B 1.6872,C 0.2508,E1 1.714,E2 534.3162} C_DIS
Startdeposition()
$VEL.CP = VEL_PRINT
LIN {X 4.6192,Y -138.365,Z 189,A -79.2338,B 1.6876,C 0.2481,E1 1.7198,E2 532.2545} C_DIS
LIN {X 8.3399,Y -138.1886,Z 189,A -77.8179,B 1.6876,C 0.2481,E1 1.7237,E2 530.8554} C_DIS
LIN {X 12.4396,Y -137.8821,Z 189,A -76.026,B 1.6878,C 0.2468,E1 1.7287,E2 529.0499} C_DIS
LIN {X 16.1624,Y -137.4933,Z 189,A -74.6475,B 1.6878,C 0.2467,E1 1.7325,E2 527.6945} C_DIS
LIN {X 20.3826,Y -136.9334,Z 189,A -72.771,B 1.6881,C 0.245,E1 1.7378,E2 525.8008} C_DIS
LIN {X 24.1498,Y -136.3173,Z 189,A -71.3667,B 1.6881,C 0.2447,E1 1.7416,E2 524.4202} C_DIS
LIN {X 28.4097,Y -135.4958,Z 189,A -69.6109,B 1.6883,C 0.2434,E1 1.7464,E2 522.669} C_DIS
LIN {X 31.6347,Y -134.7793,Z 189,A -68.2762,B 1.6885,C 0.2424,E1 1.75,E2 521.3381} C_DIS
LIN {X 34.8637,Y -133.9804,Z 189,A -66.7959,B 1.6887,C 0.2406,E1 1.7541,E2 519.8423} C_DIS
LIN {X 38.4127,Y -133.0046,Z 189,A -65.3937,B 1.6889,C 0.2397,E1 1.7579,E2 518.4561} C_DIS
LIN {X 41.8875,Y -131.9507,Z 189,A -64.2031,B 1.6889,C 0.2397,E1 1.7609,E2 517.3083} C_DIS
LIN {X 44.5436,Y -131.0805,Z 189,A -62.8737,B 1.6892,C 0.2375,E1 1.7645,E2 515.954} C_DIS
LIN {X 48.0649,Y -129.8288,Z 189,A -61.3898,B 1.6894,C 0.236,E1 1.7684,E2 514.4778} C_DIS
LIN {X 50.9598,Y -128.7218,Z 189,A -60.1392,B 1.6896,C 0.2346,E1 1.7717,E2 513.2308} C_DIS
LIN {X 54.1471,Y -127.4139,Z 189,A -58.7643,B 1.6898,C 0.233,E1 1.7752,E2 511.8621} C_DIS
LIN {X 57.6353,Y -125.8726,Z 189,A -57.3682,B 1.6899,C 0.2319,E1 1.7787,E2 510.4903} C_DIS
LIN {X 60.4634,Y -124.5407,Z 189,A -55.9072,B 1.6903,C 0.2291,E1 1.7825,E2 509.005} C_DIS
LIN {X 63.8234,Y -122.8511,Z 189,A -54.5253,B 1.6905,C 0.2278,E1 1.7859,E2 507.6464} C_DIS
LIN {X 67.4482,Y -120.9006,Z 189,A -52.7683,B 1.6909,C 0.2249,E1 1.7902,E2 505.8807} C_DIS
LIN {X 71.2597,Y -118.694,Z 189,A -51.0268,B 1.6912,C 0.2224,E1 1.7944,E2 504.1493} C_DIS
LIN {X 75.0998,Y -116.302,Z 189,A -49.3092,B 1.6915,C 0.2202,E1 1.7984,E2 502.4519} C_DIS
LIN {X 78.7034,Y -113.8946,Z 189,A -47.5349,B 1.6919,C 0.2172,E1 1.8025,E2 500.6789} C_DIS
LIN {X 82.3228,Y -111.3067,Z 189,A -45.8298,B 1.6922,C 0.2147,E1 1.8063,E2 498.9914} C_DIS
LIN {X 85.8655,Y -108.5971,Z 189,A -44.0362,B 1.6926,C 0.2116,E1 1.8103,E2 497.2037} C_DIS
LIN {X 89.4021,Y -105.7043,Z 189,A -42.2697,B 1.693,C 0.2087,E1 1.814,E2 495.453} C_DIS
LIN {X 92.697,Y -102.8274,Z 189,A -40.5811,B 1.6933,C 0.2058,E1 1.8175,E2 493.7799} C_DIS
LIN {X 95.8808,Y -99.8649,Z 189,A -38.9037,B 1.6937,C 0.2029,E1 1.8209,E2 492.1179} C_DIS
LIN {X 98.9298,Y -96.8448,Z 189,A -37.241,B 1.694,C 0.1999,E1 1.8241,E2 490.4696} C_DIS
LIN {X 101.6196,Y -94.0196,Z 189,A -35.6945,B 1.6944,C 0.1968,E1 1.8271,E2 488.9312} C_DIS
LIN {X 104.2244,Y -91.1225,Z 189,A -34.1887,B 1.6947,C 0.194,E1 1.8299,E2 487.4388} C_DIS
LIN {X 106.9144,Y -87.9518,Z 189,A -32.5518,B 1.6951,C 0.1906,E1 1.8328,E2 485.8121} C_DIS
LIN {X 109.6953,Y -84.458,Z 189,A -30.7946,B 1.6955,C 0.187,E1 1.8358,E2 484.0659} C_DIS
LIN {X 112.3566,Y -80.8839,Z 189,A -29.1136,B 1.6958,C 0.1838,E1 1.8385,E2 482.4059} C_DIS
LIN {X 114.8951,Y -77.2356,Z 189,A -27.362,B 1.6963,C 0.1799,E1 1.8413,E2 480.6649} C_DIS
LIN {X 117.3078,Y -73.5193,Z 189,A -25.644,B 1.6966,C 0.1763,E1 1.8438,E2 478.9613} C_DIS
LIN {X 119.5923,Y -69.7416,Z 189,A -23.9426,B 1.697,C 0.1726,E1 1.8462,E2 477.2756} C_DIS
LIN {X 121.7466,Y -65.909,Z 189,A -22.2562,B 1.6974,C 0.1689,E1 1.8485,E2 475.6059} C_DIS
LIN {X 123.3894,Y -62.7735,Z 189,A -21.0691,B 1.6976,C 0.1671,E1 1.8499,E2 474.4552} C_DIS
LIN {X 125.2911,Y -58.8927,Z 189,A -19.3352,B 1.698,C 0.1629,E1 1.852,E2 472.7276} C_DIS
LIN {X 126.7317,Y -55.7249,Z 189,A -18.0022,B 1.6983,C 0.1599,E1 1.8535,E2 471.408} C_DIS
LIN {X 128.0786,Y -52.5555,Z 189,A -16.5577,B 1.6986,C 0.156,E1 1.8551,E2 469.9598} C_DIS
LIN {X 129.5384,Y -48.8402,Z 189,A -15.3023,B 1.6988,C 0.1544,E1 1.8563,E2 468.7565} C_DIS
LIN {X 130.5229,Y -46.1518,Z 189,A -14.0296,B 1.6991,C 0.1506,E1 1.8575,E2 467.4713} C_DIS
LIN {X 131.6167,Y -42.9332,Z 189,A -12.7468,B 1.6994,C 0.1477,E1 1.8586,E2 466.2041} C_DIS
LIN {X 132.6254,Y -39.7078,Z 189,A -11.453,B 1.6996,C 0.1447,E1 1.8597,E2 464.9232} C_DIS
LIN {X 133.6358,Y -36.1557,Z 189,A -10.1514,B 1.6998,C 0.1421,E1 1.8606,E2 463.6508} C_DIS
LIN {X 134.3902,Y -33.2489,Z 189,A -8.8911,B 1.7001,C 0.1386,E1 1.8615,E2 462.3874} C_DIS
LIN {X 135.1478,Y -30.0215,Z 189,A -7.6237,B 1.7004,C 0.1356,E1 1.8623,E2 461.1329} C_DIS
LIN {X 135.8234,Y -26.7995,Z 189,A -6.2291,B 1.7007,C 0.1316,E1 1.8631,E2 459.7332} C_DIS
LIN {X 136.5122,Y -23.0224,Z 189,A -4.8993,B 1.7009,C 0.129,E1 1.8637,E2 458.4367} C_DIS
LIN {X 137.1616,Y -18.786,Z 189,A -3.262,B 1.7012,C 0.125,E1 1.8643,E2 456.8163} C_DIS
LIN {X 137.5599,Y -15.6042,Z 189,A -1.8998,B 1.7015,C 0.1211,E1 1.8648,E2 455.4487} C_DIS
LIN {X 137.9227,Y -11.9587,Z 189,A -0.6026,B 1.7017,C 0.1184,E1 1.8651,E2 454.1794} C_DIS
LIN {X 138.2261,Y -7.7304,Z 189,A 1.1135,B 1.702,C 0.1138,E1 1.8654,E2 452.4672} C_DIS
LIN {X 138.3801,Y -4.0759,Z 189,A 2.4102,B 1.7022,C 0.111,E1 1.8655,E2 451.1981} C_DIS
LIN {X 138.4416,Y -0.3638,Z 189,A 3.8517,B 1.7024,C 0.1074,E1 1.8655,E2 449.7682} C_DIS
LIN {X 138.408,Y 3.0729,Z 189,A 5.2356,B 1.7026,C 0.1037,E1 1.8655,E2 448.3884} C_DIS
LIN {X 138.2769,Y 6.7194,Z 189,A 6.5059,B 1.7028,C 0.1011,E1 1.8654,E2 447.1486} C_DIS
LIN {X 138.0895,Y 9.8463,Z 189,A 7.7058,B 1.7029,C 0.0982,E1 1.8651,E2 445.9605} C_DIS
LIN {X 137.6705,Y 14.5763,Z 189,A 9.5248,B 1.7032,C 0.0937,E1 1.8647,E2 444.1594} C_DIS
LIN {X 137.297,Y 17.7527,Z 189,A 10.7755,B 1.7034,C 0.0905,E1 1.8642,E2 442.9175} C_DIS
LIN {X 136.6857,Y 21.9825,Z 189,A 12.5296,B 1.7036,C 0.0857,E1 1.8635,E2 441.1644} C_DIS
LIN {X 136.0228,Y 25.7564,Z 189,A 13.7763,B 1.7037,C 0.0837,E1 1.8629,E2 439.9607} C_DIS
LIN {X 135.4958,Y 28.4097,Z 189,A 14.8927,B 1.7039,C 0.0806,E1 1.8623,E2 438.8441} C_DIS
LIN {X 134.7004,Y 31.9622,Z 189,A 16.3467,B 1.704,C 0.0769,E1 1.8614,E2 437.3962} C_DIS
LIN {X 133.5497,Y 36.4786,Z 189,A 18.0766,B 1.7042,C 0.073,E1 1.8602,E2 435.691} C_DIS
LIN {X 132.6254,Y 39.7078,Z 189,A 19.4547,B 1.7044,C 0.0693,E1 1.8591,E2 434.3139} C_DIS
LIN {X 131.4459,Y 43.4462,Z 189,A 20.8832,B 1.7044,C 0.0662,E1 1.8579,E2 432.9093} C_DIS
LIN {X 130.3195,Y 46.716,Z 189,A 22.199,B 1.7046,C 0.0632,E1 1.8567,E2 431.6076} C_DIS
LIN {X 129.3436,Y 49.3603,Z 189,A 23.3958,B 1.7047,C 0.0599,E1 1.8555,E2 430.4066} C_DIS
LIN {X 127.9344,Y 52.9009,Z 189,A 24.7203,B 1.7048,C 0.0575,E1 1.8541,E2 429.1135} C_DIS
LIN {X 126.7278,Y 55.7341,Z 189,A 25.9798,B 1.7049,C 0.0542,E1 1.8527,E2 427.8555} C_DIS
LIN {X 125.2911,Y 58.8927,Z 189,A 27.2669,B 1.7049,C 0.0515,E1 1.8512,E2 426.5868} C_DIS
LIN {X 123.769,Y 62.0279,Z 189,A 28.711,B 1.7051,C 0.0478,E1 1.8494,E2 425.142} C_DIS
LIN {X 121.813,Y 65.7853,Z 189,A 30.3233,B 1.7051,C 0.0443,E1 1.8473,E2 423.5469} C_DIS
LIN {X 119.5923,Y 69.7416,Z 189,A 32.0974,B 1.7053,C 0.0403,E1 1.8449,E2 421.7853} C_DIS
LIN {X 117.3078,Y 73.5193,Z 189,A 33.8069,B 1.7053,C 0.0366,E1 1.8424,E2 420.0901} C_DIS
LIN {X 114.8951,Y 77.2356,Z 189,A 35.5201,B 1.7054,C 0.033,E1 1.8398,E2 418.3916} C_DIS
LIN {X 112.3566,Y 80.8839,Z 189,A 37.2348,B 1.7055,C 0.0294,E1 1.837,E2 416.692} C_DIS
LIN {X 109.6953,Y 84.458,Z 189,A 38.9669,B 1.7055,C 0.0258,E1 1.8341,E2 414.9735} C_DIS
LIN {X 106.9144,Y 87.9518,Z 189,A 40.5867,B 1.7056,C 0.0231,E1 1.8313,E2 413.3817} C_DIS
LIN {X 104.2599,Y 91.0818,Z 189,A 42.2281,B 1.7056,C 0.0196,E1 1.8283,E2 411.7471} C_DIS
LIN {X 101.4051,Y 94.2499,Z 189,A 43.8844,B 1.7056,C 0.0165,E1 1.8252,E2 410.104} C_DIS
LIN {X 98.5249,Y 97.2577,Z 189,A 45.5291,B 1.7057,C 0.0133,E1 1.822,E2 408.4689} C_DIS
LIN {X 95.7468,Y 99.9929,Z 189,A 47.0256,B 1.7057,C 0.0106,E1 1.8191,E2 406.9866} C_DIS
LIN {X 92.697,Y 102.8274,Z 189,A 48.6745,B 1.7057,C 0.0076,E1 1.8157,E2 405.3467} C_DIS
LIN {X 89.3584,Y 105.7415,Z 189,A 50.4112,B 1.7057,C 0.0046,E1 1.812,E2 403.6218} C_DIS
LIN {X 85.8655,Y 108.5971,Z 189,A 52.2181,B 1.7057,C 0.0014,E1 1.8081,E2 401.8222} C_DIS
LIN {X 82.2321,Y 111.3733,Z 189,A 53.9411,B 1.7057,C -0.0011,E1 1.8043,E2 400.1199} C_DIS
LIN {X 78.7034,Y 113.8946,Z 189,A 55.7158,B 1.7057,C -0.0042,E1 1.8002,E2 398.3476} C_DIS
LIN {X 75.0136,Y 116.358,Z 189,A 57.4375,B 1.7057,C -0.0067,E1 1.7962,E2 396.64} C_DIS
LIN {X 71.2597,Y 118.694,Z 189,A 59.1633,B 1.7057,C -0.0091,E1 1.7921,E2 394.9269} C_DIS
LIN {X 67.4482,Y 120.9006,Z 189,A 60.9454,B 1.7057,C -0.0118,E1 1.7878,E2 393.1498} C_DIS
LIN {X 63.3629,Y 123.0893,Z 189,A 62.579,B 1.7057,C -0.0131,E1 1.7838,E2 391.5506} C_DIS
LIN {X 60.4634,Y 124.5407,Z 189,A 64.0602,B 1.7057,C -0.0158,E1 1.7801,E2 390.053} C_DIS
LIN {X 57.3161,Y 126.0202,Z 189,A 65.3342,B 1.7057,C -0.0169,E1 1.7769,E2 388.799} C_DIS
LIN {X 53.6719,Y 127.6124,Z 189,A 66.9241,B 1.7057,C -0.0188,E1 1.7728,E2 387.216} C_DIS
LIN {X 50.3976,Y 128.9404,Z 189,A 68.111,B 1.7057,C -0.0192,E1 1.7698,E2 386.0623} C_DIS
LIN {X 47.7575,Y 129.944,Z 189,A 69.4522,B 1.7057,C -0.0215,E1 1.7662,E2 384.7009} C_DIS
LIN {X 44.5436,Y 131.0805,Z 189,A 70.9518,B 1.7057,C -0.0235,E1 1.7622,E2 383.1909} C_DIS
LIN {X 40.7543,Y 132.3051,Z 189,A 72.4095,B 1.7056,C -0.0244,E1 1.7584,E2 381.7563} C_DIS
LIN {X 37.5261,Y 133.2568,Z 189,A 73.7601,B 1.7056,C -0.0255,E1 1.7548,E2 380.411} C_DIS
LIN {X 34.8637,Y 133.9804,Z 189,A 75.0061,B 1.7056,C -0.0271,E1 1.7514,E2 379.1531} C_DIS
LIN {X 31.068,Y 134.9088,Z 189,A 76.4424,B 1.7056,C -0.0277,E1 1.7475,E2 377.7387} C_DIS
LIN {X 27.844,Y 135.6109,Z 189,A 77.5665,B 1.7056,C -0.0277,E1 1.7445,E2 376.6436} C_DIS
LIN {X 24.6708,Y 136.224,Z 189,A 79.09,B 1.7056,C -0.0296,E1 1.7402,E2 375.0985} C_DIS
LIN {X 21.4204,Y 136.7727,Z 189,A 80.4138,B 1.7055,C -0.0303,E1 1.7366,E2 373.7799} C_DIS
LIN {X 17.1931,Y 137.3704,Z 189,A 82.1466,B 1.7055,C -0.0313,E1 1.7318,E2 372.0518} C_DIS
LIN {X 13.4645,Y 137.7837,Z 189,A 83.4693,B 1.7055,C -0.0312,E1 1.7282,E2 370.7567} C_DIS
LIN {X 10.8646,Y 138.0151,Z 189,A 84.7346,B 1.7055,C -0.0324,E1 1.7246,E2 369.47} C_DIS
LIN {X 7.7304,Y 138.2261,Z 189,A 86.1635,B 1.7055,C -0.0335,E1 1.7205,E2 368.0263} C_DIS
LIN {X 4.0164,Y 138.3818,Z 189,A 87.5581,B 1.7055,C -0.0335,E1 1.7167,E2 366.6493} C_DIS
LIN {X -0.5386,Y 138.4391,Z 189,A 89.206,B 1.7055,C -0.0331,E1 1.7121,E2 365.0302} C_DIS
LIN {X -3.6614,Y 138.3916,Z 189,A 90.4751,B 1.7055,C -0.0332,E1 1.7086,E2 363.7644} C_DIS
LIN {X -6.7194,Y 138.2769,Z 189,A 91.9569,B 1.7055,C -0.0342,E1 1.7044,E2 362.2578} C_DIS
LIN {X -10.0262,Y 138.0763,Z 189,A 93.353,B 1.7055,C -0.0344,E1 1.7004,E2 360.8593} C_DIS
LIN {X -13.4645,Y 137.7837,Z 189,A 94.8127,B 1.7055,C -0.0344,E1 1.6964,E2 359.3966} C_DIS
LIN {X -17.7527,Y 137.297,Z 189,A 96.3423,B 1.7055,C -0.0335,E1 1.6922,E2 357.898} C_DIS
LIN {X -20.3826,Y 136.9334,Z 189,A 97.6585,B 1.7055,C -0.034,E1 1.6885,E2 356.5568} C_DIS
LIN {X -24.1498,Y 136.3173,Z 189,A 99.2519,B 1.7055,C -0.0337,E1 1.6841,E2 354.9624} C_DIS
LIN {X -28.4097,Y 135.4958,Z 189,A 101.0663,B 1.7055,C -0.0332,E1 1.6791,E2 353.1468} C_DIS
LIN {X -31.6347,Y 134.7793,Z 189,A 102.4517,B 1.7055,C -0.0328,E1 1.6753,E2 351.76} C_DIS
LIN {X -34.8637,Y 133.9804,Z 189,A 103.8494,B 1.7055,C -0.0322,E1 1.6715,E2 350.3605} C_DIS
LIN {X -38.0935,Y 133.0981,Z 189,A 105.3431,B 1.7055,C -0.0318,E1 1.6674,E2 348.8548} C_DIS
LIN {X -41.5889,Y 132.0461,Z 189,A 106.6929,B 1.7055,C -0.0305,E1 1.6638,E2 347.5248} C_DIS
LIN {X -44.5436,Y 131.0805,Z 189,A 108.1136,B 1.7055,C -0.03,E1 1.66,E2 346.089} C_DIS
LIN {X -47.7575,Y 129.944,Z 189,A 109.6907,B 1.7055,C -0.0294,E1 1.6558,E2 344.4929} C_DIS
LIN {X -51.4223,Y 128.5354,Z 189,A 111.0344,B 1.7055,C -0.0274,E1 1.6524,E2 343.1834} C_DIS
LIN {X -54.5283,Y 127.2491,Z 189,A 112.4965,B 1.7055,C -0.0264,E1 1.6486,E2 341.7138} C_DIS
LIN {X -57.3161,Y 126.0202,Z 189,A 114.099,B 1.7055,C -0.026,E1 1.6444,E2 340.0716} C_DIS
LIN {X -60.4634,Y 124.5407,Z 189,A 115.4393,B 1.7055,C -0.0243,E1 1.641,E2 338.7439} C_DIS
LIN {X -63.5857,Y 122.9759,Z 189,A 117.0094,B 1.7056,C -0.0231,E1 1.6371,E2 337.1598} C_DIS
LIN {X -67.4482,Y 120.9006,Z 189,A 118.9395,B 1.7056,C -0.0213,E1 1.6323,E2 335.2171} C_DIS
LIN {X -71.2597,Y 118.694,Z 189,A 120.8345,B 1.7056,C -0.0192,E1 1.6277,E2 333.3145} C_DIS
LIN {X -75.0136,Y 116.358,Z 189,A 122.7354,B 1.7056,C -0.0169,E1 1.6232,E2 331.4063} C_DIS
LIN {X -78.7034,Y 113.8946,Z 189,A 124.6602,B 1.7057,C -0.0145,E1 1.6187,E2 329.472} C_DIS
LIN {X -82.3228,Y 111.3067,Z 189,A 126.5391,B 1.7057,C -0.0119,E1 1.6145,E2 327.5898} C_DIS
LIN {X -85.8655,Y 108.5971,Z 189,A 128.527,B 1.7057,C -0.0093,E1 1.61,E2 325.5861} C_DIS
LIN {X -89.3255,Y 105.7694,Z 189,A 130.3447,B 1.7057,C -0.0062,E1 1.6061,E2 323.7734} C_DIS
LIN {X -92.0301,Y 103.4248,Z 189,A 131.9851,B 1.7057,C -0.0039,E1 1.6026,E2 322.1148} C_DIS
LIN {X -94.904,Y 100.7932,Z 189,A 133.6625,B 1.7057,C -0.0012,E1 1.5992,E2 320.4306} C_DIS
LIN {X -97.8933,Y 97.8933,Z 189,A 135.5505,B 1.7057,C 0.0017,E1 1.5954,E2 318.524} C_DIS
LIN {X -101.0091,Y 94.6751,Z 189,A 137.4807,B 1.7057,C 0.0052,E1 1.5916,E2 316.5858} C_DIS
LIN {X -103.8093,Y 91.595,Z 189,A 139.2779,B 1.7057,C 0.0084,E1 1.5883,E2 314.7807} C_DIS
LIN {X -106.5445,Y 88.3985,Z 189,A 141.14,B 1.7057,C 0.0118,E1 1.5849,E2 312.905} C_DIS
LIN {X -109.1486,Y 85.1634,Z 189,A 143.0517,B 1.7057,C 0.0152,E1 1.5815,E2 310.971} C_DIS
LIN {X -111.8341,Y 81.6049,Z 189,A 144.9737,B 1.7057,C 0.0191,E1 1.5783,E2 309.0409} C_DIS
LIN {X -114.3974,Y 77.9709,Z 189,A 146.9449,B 1.7057,C 0.023,E1 1.5752,E2 307.0549} C_DIS
LIN {X -116.8354,Y 74.2677,Z 189,A 148.9644,B 1.7056,C 0.027,E1 1.5721,E2 305.0139} C_DIS
LIN {X -119.1458,Y 70.5018,Z 189,A 150.9297,B 1.7055,C 0.0311,E1 1.5692,E2 303.0331} C_DIS
LIN {X -121.3262,Y 66.6796,Z 189,A 152.7612,B 1.7055,C 0.0354,E1 1.5667,E2 301.2016} C_DIS
LIN {X -122.9759,Y 63.5857,Z 189,A 154.4808,B 1.7053,C 0.0387,E1 1.5644,E2 299.4496} C_DIS
LIN {X -124.5407,Y 60.4634,Z 189,A 155.8856,B 1.7053,C 0.0423,E1 1.5627,E2 298.0509} C_DIS
LIN {X -126.0202,Y 57.3161,Z 189,A 157.4409,B 1.7052,C 0.0458,E1 1.5609,E2 296.4822} C_DIS
LIN {X -127.4139,Y 54.1471,Z 189,A 158.9904,B 1.7051,C 0.0493,E1 1.5591,E2 294.9191} C_DIS
LIN {X -128.8279,Y 50.6869,Z 189,A 160.7149,B 1.7049,C 0.0532,E1 1.5573,E2 293.1734} C_DIS
LIN {X -130.0913,Y 47.3489,Z 189,A 162.0913,B 1.7049,C 0.0571,E1 1.556,E2 291.8106} C_DIS
LIN {X -131.0805,Y 44.5436,Z 189,A 163.6015,B 1.7047,C 0.0601,E1 1.5546,E2 290.2664} C_DIS
LIN {X -132.1317,Y 41.3212,Z 189,A 165.284,B 1.7046,C 0.0636,E1 1.5531,E2 288.5496} C_DIS
LIN {X -133.2568,Y 37.5261,Z 189,A 166.9027,B 1.7044,C 0.068,E1 1.5519,E2 286.9343} C_DIS
LIN {X -133.9804,Y 34.8637,Z 189,A 168.1443,B 1.7043,C 0.071,E1 1.551,E2 285.681} C_DIS
LIN {X -134.7793,Y 31.6347,Z 189,A 169.7393,B 1.7041,C 0.0746,E1 1.5499,E2 284.0592} C_DIS
LIN {X -135.6109,Y 27.844,Z 189,A 171.3499,B 1.7039,C 0.0789,E1 1.549,E2 282.4491} C_DIS
LIN {X -136.2317,Y 24.628,Z 189,A 172.8641,B 1.7038,C 0.0826,E1 1.5482,E2 280.9155} C_DIS
LIN {X -136.7727,Y 21.4204,Z 189,A 174.3298,B 1.7036,C 0.0862,E1 1.5475,E2 279.4354} C_DIS
LIN {X -137.3704,Y 17.1931,Z 189,A 176.2556,B 1.7033,C 0.091,E1 1.5468,E2 277.4905} C_DIS
LIN {X -137.7837,Y 13.4645,Z 189,A 177.956,B 1.7031,C 0.0952,E1 1.5463,E2 275.772} C_DIS
LIN {X -138.1297,Y 9.2948,Z 189,A 179.8345,B 1.7028,C 0.0999,E1 1.5459,E2 273.8758} C_DIS
LIN {X -138.3257,Y 5.6263,Z 189,A -178.509,B 1.7026,C 0.1041,E1 1.5457,E2 272.2027} C_DIS
LIN {X -138.4336,Y 1.533,Z 189,A -176.5869,B 1.7023,C 0.1087,E1 1.5456,E2 270.2522} C_DIS
LIN {X -138.4198,Y -2.3643,Z 189,A -174.8412,B 1.702,C 0.1131,E1 1.5456,E2 268.4901} C_DIS
LIN {X -138.3045,Y -6.1718,Z 189,A -173.0077,B 1.7017,C 0.1174,E1 1.5458,E2 266.6242} C_DIS
LIN {X -138.0895,Y -9.8463,Z 189,A -171.5054,B 1.7014,C 0.1216,E1 1.5461,E2 265.1254} C_DIS
LIN {X -137.6705,Y -14.5763,Z 189,A -169.3564,B 1.701,C 0.127,E1 1.5467,E2 262.9535} C_DIS
LIN {X -137.2823,Y -17.8651,Z 189,A -167.8716,B 1.7008,C 0.1307,E1 1.5472,E2 261.4544} C_DIS
LIN {X -136.6857,Y -21.9825,Z 189,A -165.807,B 1.7004,C 0.1351,E1 1.5481,E2 259.3458} C_DIS
LIN {X -135.8234,Y -26.7995,Z 189,A -163.6864,B 1.7,C 0.1406,E1 1.5492,E2 257.2136} C_DIS
LIN {X -135.0732,Y -30.3481,Z 189,A -162.0602,B 1.6996,C 0.1446,E1 1.5502,E2 255.5715} C_DIS
LIN {X -134.2462,Y -33.8162,Z 189,A -160.7567,B 1.6993,C 0.1487,E1 1.551,E2 254.2915} C_DIS
LIN {X -133.5497,Y -36.4786,Z 189,A -159.1152,B 1.699,C 0.1513,E1 1.5523,E2 252.5839} C_DIS
LIN {X -132.4821,Y -40.1761,Z 189,A -157.5193,B 1.6987,C 0.1555,E1 1.5535,E2 250.9882} C_DIS
LIN {X -131.6167,Y -42.9332,Z 189,A -156.2468,B 1.6984,C 0.1586,E1 1.5546,E2 249.7061} C_DIS
LIN {X -130.5229,Y -46.1518,Z 189,A -154.7184,B 1.698,C 0.1621,E1 1.556,E2 248.162} C_DIS
LIN {X -129.3436,Y -49.3603,Z 189,A -153.183,B 1.6977,C 0.1657,E1 1.5576,E2 246.6111} C_DIS
LIN {X -128.0786,Y -52.5555,Z 189,A -151.641,B 1.6974,C 0.1692,E1 1.5592,E2 245.0536} C_DIS
LIN {X -126.7278,Y -55.7341,Z 189,A -150.0933,B 1.697,C 0.1726,E1 1.5609,E2 243.4905} C_DIS
LIN {X -125.2911,Y -58.8927,Z 189,A -148.4447,B 1.6967,C 0.1759,E1 1.5629,E2 241.8138} C_DIS
LIN {X -123.6124,Y -62.3354,Z 189,A -146.8804,B 1.6963,C 0.1798,E1 1.5648,E2 240.2528} C_DIS
LIN {X -122.0158,Y -65.4078,Z 189,A -145.1839,B 1.6959,C 0.1829,E1 1.5671,E2 238.5212} C_DIS
LIN {X -119.7474,Y -69.4738,Z 189,A -143.1623,B 1.6955,C 0.1873,E1 1.5699,E2 236.4873} C_DIS
LIN {X -117.472,Y -73.2555,Z 189,A -141.1988,B 1.695,C 0.1913,E1 1.5728,E2 234.5057} C_DIS
LIN {X -115.2147,Y -76.7568,Z 189,A -139.295,B 1.6946,C 0.1949,E1 1.5758,E2 232.5779} C_DIS
LIN {X -112.5385,Y -80.6295,Z 189,A -137.2629,B 1.6941,C 0.199,E1 1.579,E2 230.5348} C_DIS
LIN {X -110.0468,Y -83.9984,Z 189,A -135.3561,B 1.6937,C 0.2024,E1 1.5823,E2 228.6047} C_DIS
LIN {X -107.1131,Y -87.7087,Z 189,A -133.2881,B 1.6933,C 0.2063,E1 1.5859,E2 226.5219} C_DIS
LIN {X -104.2244,Y -91.1225,Z 189,A -131.3543,B 1.6928,C 0.2098,E1 1.5895,E2 224.577} C_DIS
LIN {X -101.2415,Y -94.4256,Z 189,A -129.3947,B 1.6924,C 0.2131,E1 1.5932,E2 222.6015} C_DIS
LIN {X -98.5249,Y -97.2577,Z 189,A -127.6461,B 1.6921,C 0.2158,E1 1.5967,E2 220.8359} C_DIS
LIN {X -95.7468,Y -99.9929,Z 189,A -125.9677,B 1.6917,C 0.2186,E1 1.6001,E2 219.1486} C_DIS
LIN {X -92.697,Y -102.8274,Z 189,A -124.0958,B 1.6914,C 0.2212,E1 1.604,E2 217.2563} C_DIS
LIN {X -89.3255,Y -105.7694,Z 189,A -122.1776,B 1.691,C 0.2241,E1 1.6081,E2 215.3289} C_DIS
LIN {X -85.8655,Y -108.5971,Z 189,A -120.1889,B 1.6906,C 0.2267,E1 1.6125,E2 213.3209} C_DIS
LIN {X -82.3228,Y -111.3067,Z 189,A -118.2646,B 1.6903,C 0.2293,E1 1.6168,E2 211.3857} C_DIS
LIN {X -78.7034,Y -113.8946,Z 189,A -116.3372,B 1.69,C 0.2316,E1 1.6212,E2 209.4462} C_DIS
LIN {X -75.0136,Y -116.358,Z 189,A -114.4397,B 1.6897,C 0.2339,E1 1.6257,E2 207.5401} C_DIS
LIN {X -71.2597,Y -118.694,Z 189,A -112.5761,B 1.6894,C 0.2361,E1 1.6302,E2 205.6716} C_DIS
LIN {X -67.4482,Y -120.9006,Z 189,A -110.6423,B 1.6891,C 0.2379,E1 1.6349,E2 203.722} C_DIS
LIN {X -63.5857,Y -122.9759,Z 189,A -108.7861,B 1.6888,C 0.2397,E1 1.6395,E2 201.8598} C_DIS
LIN {X -60.4634,Y -124.5407,Z 189,A -107.4018,B 1.6886,C 0.2413,E1 1.643,E2 200.4838} C_DIS
LIN {X -56.8719,Y -126.2189,Z 189,A -105.7806,B 1.6884,C 0.2429,E1 1.6471,E2 198.8649} C_DIS
LIN {X -53.6743,Y -127.6114,Z 189,A -104.4276,B 1.6882,C 0.2444,E1 1.6506,E2 197.5243} C_DIS
LIN {X -50.9598,Y -128.7218,Z 189,A -102.9945,B 1.6882,C 0.2447,E1 1.6544,E2 196.0603} C_DIS
LIN {X -47.7575,Y -129.944,Z 189,A -101.4235,B 1.6881,C 0.2452,E1 1.6586,E2 194.4676} C_DIS
LIN {X -44.2396,Y -131.1817,Z 189,A -100.0926,B 1.6878,C 0.2469,E1 1.662,E2 193.166} C_DIS
LIN {X -41.3212,Y -132.1317,Z 189,A -98.6829,B 1.6878,C 0.2472,E1 1.6658,E2 191.7364} C_DIS
LIN {X -38.0935,Y -133.0981,Z 189,A -97.1435,B 1.6878,C 0.2474,E1 1.67,E2 190.1762} C_DIS
LIN {X -34.2771,Y -134.1292,Z 189,A -95.835,B 1.6875,C 0.2493,E1 1.6735,E2 188.9131} C_DIS
LIN {X -31.6347,Y -134.7793,Z 189,A -94.4751,B 1.6875,C 0.2489,E1 1.6773,E2 187.5201} C_DIS
LIN {X -27.9757,Y -135.5841,Z 189,A -93.0738,B 1.6874,C 0.25,E1 1.6811,E2 186.1392} C_DIS
LIN {X -25.1913,Y -136.1309,Z 189,A -91.5764,B 1.6874,C 0.249,E1 1.6853,E2 184.596} C_DIS
LIN {X -21.4204,Y -136.7727,Z 189,A -90.1423,B 1.6874,C 0.2499,E1 1.6892,E2 183.1822} C_DIS
Enddeposition()
END
